(* PLC project IndraLogic.project, IndraLogic indralogic *)
(* stored: creationDateTime 2023-05-04T16:21:11.22622, modificationDateTime 2023-04-06T09:56:36 *)

{attribute 'symbol' := 'none'}
TYPE ST_ComBasketRotation : STRUCT
  fBasketRotationSpeed : REAL;  (* Drehzahl 0 <= x <= 4 l/min *)
  diagCodeBasketRotation : IL_INLN_DIAG_CODE;  (* Sensor-Diagnose: Temperatur *)
END_STRUCT;
END_TYPE

{attribute 'symbol' := 'readwrite'}
TYPE ST_TankErrorState : STRUCT
  bErrorTankLevelLow : BOOL;
  bErrorTankLevelFull : BOOL;
  bErrorFreshWaterSupply : BOOL;
  bErrorTankTemperatureCriticalLow : BOOL;
  bErrorTankTemperatureCriticalHigh : BOOL;
END_STRUCT;
END_TYPE

{attribute 'symbol' := 'none'}
TYPE ST_PowerMeasurementUMG96RM : STRUCT
  modeReturn : INT;  (* Die genaue Konfiguration ist dem Handbuch zu Janitza UMG96RM-P (ab S.82) zu entnehmen *)
  value : ARRAY[0..26] OF REAL;
  count : INT := 27;
  StromGes : REAL;
  WirkleistungGes : REAL;
  BlindleistungGes : REAL;
  Frequenz : REAL;
END_STRUCT;
END_TYPE

{attribute 'symbol' := 'readwrite'}
TYPE ST_SetKEAProgramManual : STRUCT
  fTankTemperatureSetPointManual : REAL;  (* Bereich: 30...75°C *)
  fTankHeaterHysteresisWidthManual : REAL;  (* Definiert Range der Tankheizung *)
  fAirHeatingTemperatureSetPointManual : REAL;  (* Bereich: 50...110°C *)
  fTemperatureLimitLowerWorking : REAL;  (* minimal temperature to start process *)
  fTemperatureLimitUpperWorking : REAL;  (* maximal temperature to start process *)
  nDurationSprayCleaningManual : INT;  (* Bereich: 0...300 Sekunden - Zeit für Schrittkette *)
  nDurationDrippingManual : INT;  (* Bereich: 0...300 Sekunden - Zeit für Schrittkette *)
  nDurationSuctionManual : INT;  (* Bereich: 0...300 Sekunden - Zeit für Schrittkette *)
  nDurationBlowingManual : INT;  (* Bereich: 0...300 Sekunden - Zeit für Schrittkette *)
  nDurationConvectionDryingManual : INT;  (* Bereich: 0...300 Sekunden - Zeit für Schrittkette *)
  bProgramWithBasketRotationManual : BOOL;
  bProgramWithBasketRotation : BOOL;  (* Keine Korbrotation *)
  sTypeWorkpiece : STRING;
  fMassWorkpiece : REAL;  (* mass in kg *)
END_STRUCT;
END_TYPE

{attribute 'symbol' := 'readwrite'}
TYPE ST_KEALocalSetParameters : STRUCT
  nSelectProgram : INT;
  bSetSelectedProgram : BOOL;
  bResetErrors : BOOL;
  bOpenDoor : BOOL;
  nWorkpieces : INT;
END_STRUCT;
END_TYPE

{attribute 'symbol' := 'readwrite'}
TYPE ST_StoreEnergyInherentlyState : STRUCT
  fNominalLoad : REAL;  (* static; module's nominal load *)
  sMachineStateCorrelation : STRING;  (* static; machine states in which the module can be used as inherent energy storage: oﬀ , standby , operational or working *)
  sProcessStepCorrelation : STRING;  (* static; process steps in which the module is active *)
  sPowerUnit : STRING;  (* static; unit of nominal load and power consumption *)
  bOperatingPoint : BOOL;  (* dynamic; module's switching state *)
  fProcessValue : REAL;  (* dynamic; process value influenced by the module *)
  aFlexibilityLimits : ARRAY[1..2] OF REAL;  (* dynamic; upper and lower limits in which the energy-ﬂexible module may operate *)
  sProcessValueUnit : STRING;  (* static; unit of process value and flexibility limits *)
END_STRUCT;
END_TYPE

{attribute 'symbol' := 'readwrite'}
TYPE ST_CleaningChamberState : STRUCT
  bPumpSupplyStatusOn : BOOL;
  bRotationBasketStatusOn : BOOL;
  bRotationBasketDirectionOfRotation : BOOL;
  bRotationNoozleFrameStatusOn : BOOL;
  bExhaustAirFanStatusOn : BOOL;
  bBlastNoozleTopStatusOn : BOOL;
  bBlastNoozleBottomStatusOn : BOOL;
  bProtectiveDoorLoadingOpen : BOOL;
END_STRUCT;
END_TYPE

{attribute 'symbol' := 'readwrite'}
TYPE ST_InterruptProcessState : STRUCT
  stepEnergyConsumption : ST_StepEnergyConsumption;  (* static; shows total energy consumption per step for all steps that can be interrupted *)
  sEnergyUnit : STRING;  (* static; unit of energy consumption *)
  fMachinePowerConsumption : REAL;  (* dynamic; current power consumption of the whole machine *)
  stepPowerConsumption : ST_StepPowerConsumption;  (* static; shows total power consumption per step for all energy relevant steps *)
  sPowerUnit : STRING;  (* static; unit of nmachine power consumption *)
  stepDuration : ST_StepDuration;
  sMachineState : STRING;  (* dynamic; shows current machine state: oﬀ , standby , operational or working *)
  fInterruptionCountdown : REAL;  (* dynamic; shows duration until the next position for process interruption is reached *)
  fInterruptionCountdownUnit : STRING;  (* static; unit of interruption countdown *)
  nInterruptedState : E_KEAOperatingState;  (* last state before interruption *)
END_STRUCT;
END_TYPE

{attribute 'qualified_only'}
{attribute 'strict'}
TYPE E_SystemControlState : (automatic := 0, algorithm := 1, manual := 2);
END_TYPE

{attribute 'qualified_only'}
{attribute 'strict'}
TYPE E_SystemOperatingState : (standby := 0, rampUp := 1, rampDown := 2, operational := 3, working := 4);
END_TYPE

{attribute 'symbol' := 'readwrite'}
TYPE ST_Control : STRUCT
  bSetStatusOnAlgorithm : BOOL;  (* turn actor on *)
  bSetStatusOnManual : BOOL;  (* turn actor on *)
  bAlgorithmModeActivated : BOOL;  (* activate algorithm control *)
  bManualModeActivated : BOOL;  (* activate manual control *)
END_STRUCT;
END_TYPE

{attribute 'symbol' := 'readwrite'}
TYPE ST_ControlState : STRUCT
  bStatusOn : BOOL;  (* status on / off *)
  sAccessMode : STRING;  (* current access mode as string *)
  nAccessmode : E_SystemControlState;  (* current access mode (1 = automatic, 2 = algorihm, 3 = manual) *)
END_STRUCT;
END_TYPE

{attribute 'symbol' := 'readwrite'}
TYPE ST_SensorState : STRUCT
  fValue : REAL;  (* status on / off *)
  sUnit : STRING;  (* current unit of sensor value *)
END_STRUCT;
END_TYPE

{attribute 'symbol' := 'readwrite'}
TYPE ST_SetPointState : STRUCT
  fOperatingPoint : REAL;  (* current operating point *)
  fSetPoint : REAL;  (* current set point *)
  sSetPointUnit : STRING;  (* current set point unit *)
  sOperatingPointUnit : STRING;  (* current operating point unit *)
  aSetPointLimits : ARRAY[1..2] OF REAL;  (* lower and upper limit of setpoint *)
END_STRUCT;
END_TYPE

{attribute 'symbol' := 'readwrite'}
TYPE ST_SetSetPoint : STRUCT
  fSetPointAlgorithm : REAL;  (* set setpoint in percent 0.0 - 100.0 *)
  fSetPointManual : REAL;  (* set setpoint in percent 0.0 - 100.0 *)
END_STRUCT;
END_TYPE

{attribute 'symbol' := 'readwrite'}
TYPE ST_SystemState : STRUCT
  sOperatingState : STRING;  (* operating state (standby, operational, working) *)
  nOperatingState : E_SystemOperatingState;  (* operating state (standby, operational, working) *)
  bError : BOOL;  (* true if there is an error in any system component *)
END_STRUCT;
END_TYPE

{attribute 'symbol' := 'readwrite'}
TYPE ST_InletAirHeatingErrorState : STRUCT
  bInletAirShutOffValveOpeningError : BOOL;
  bInletAirShutOffValveClosingError : BOOL;
  bInletAirShutOffValveSensorsError : BOOL;
  bInletAirFanError : BOOL;
  bAirSupplyTempSensorError : BOOL;
  bErrorAirTemperatureCriticalLow : BOOL;
  bErrorAirTemperatureCriticalHigh : BOOL;
END_STRUCT;
END_TYPE

{attribute 'symbol' := 'readwrite'}
TYPE ST_TempSensorState : STRUCT
  {attribute 'symbol' := 'none'}
  senTdiag : IL_INLN_DIAG_CODE;  (* Sensor-Diagnose: Temperatur *)
END_STRUCT;
END_TYPE

{attribute 'symbol' := 'readwrite'}
TYPE ST_TankState : STRUCT
  bTankHeatingOn : BOOL;
  bSupplyFreshWaterOn : BOOL;
  bOilSeparationOn : BOOL;
  fTankTemperature : REAL;
  bFilterMonitor : BOOL;
  bTankLevelMin : BOOL;
  bTankLevelNominal : BOOL;
  bTankLevelMax : BOOL;
  bOilSeparationLevelMax : BOOL;
  bDemineralOk : BOOL;
  fTankHeaterHysteresisWidth : REAL;
  fTemperatureLimitLowerWorking : REAL;
  fTemperatureLimitUpperWorking : REAL;
  fTemperatureLimitLowerCritical : REAL;
  fTemperatureLimitUpperCritical : REAL;
  sTemperatureUnit : STRING;
  fCleaningFluidSpecificHeatCapacity : REAL;
  sCleaningFluidSpecificHeatCapacityUnit : STRING;
  fCleaningFluidDensity : REAL;
  sCleaningFluidDensityUnit : STRING;
  fTankVolume : REAL;
  sTankVolumeUnit : STRING;
END_STRUCT;
END_TYPE

{attribute 'symbol' := 'readwrite'}
TYPE ST_InletAirHeatingState : STRUCT
  fAirSupplyTemperature : REAL;
  bInletAirShutOffValveOpen : BOOL;
  bInletAirShutOffValveClosed : BOOL;
  bAirSupplyTempOk : BOOL;
  bAirSupplyFlowOk : BOOL;
  fTemperatureLimitLowerCritical : REAL;
  fTemperatureLimitUpperCritical : REAL;
  bInletAirFanStatusOn : BOOL;
END_STRUCT;
END_TYPE

{attribute 'symbol' := 'none'}
TYPE ST_KEADefaultParameters : STRUCT
  tBlastNoozlesPulseDuration : TIME := TIME#200ms;  (* Bereich: 0,2...1,0 Sekunden *)
  tBlastNoozlesPulsePeriod : TIME := TIME#700ms;  (* Bereich: 0,2...1,0 Sekunden *)
  tBasketHomeingDuration : TIME := TIME#500ms;  (* Bereich: 0,000...2,000 Sekunden - in Millisekunden verarbeiten *)
  fBasketRotationSpeed : REAL := 3;  (* Bereich: 1.5...4.0 l/min - Vorgabe für Frequenzumrichter *)
  tMaxDurationExhaustFanOn : TIME := TIME#1m0s0ms;  (* Zeitliche Begrenzung Abluftgebläse wenn Tür offen *)
END_STRUCT;
END_TYPE

{attribute 'qualified_only'}
TYPE E_KEAOperatingState : (standby := 0, rampUp := 1, operational := 2, sprayCleaning := 3, dripping := 4, suction := 5, blowing := 6, convectionDrying := 7, homing := 8, interruption := 9, break := 10, error := 11);
END_TYPE

{attribute 'symbol' := 'readwrite'}
TYPE ST_KEAProgramState : STRUCT
  sActiveProgram : STRING;
  fTankTemperatureSetPoint : REAL;  (* Bereich: 30...75°C *)
  fTankHeaterHysteresisWidth : REAL;  (* Definiert Range der Tankheizung *)
  fTemperatureLimitLowerWorking : REAL;  (* minimal temperature to start process *)
  fTemperatureLimitUpperWorking : REAL;  (* maximal temperature to start process *)
  fAirHeatingTemperatureSetPoint : REAL;  (* Bereich: 50...110°C *)
  nDurationSprayCleaning : INT;  (* Bereich: 0...300 Sekunden - Zeit für Schrittkette *)
  nDurationDripping : INT;  (* Bereich: 0...300 Sekunden - Zeit für Schrittkette *)
  nDurationSuction : INT;  (* Bereich: 0...300 Sekunden - Zeit für Schrittkette *)
  nDurationBlowing : INT;  (* Bereich: 0...300 Sekunden - Zeit für Schrittkette *)
  nDurationConvectionDrying : INT;  (* Bereich: 0...300 Sekunden - Zeit für Schrittkette *)
  sDurationUnit : STRING;  (* duration unit = seconds *)
  bProgramWithBasketRotation : BOOL;
  sTypeWorkpiece : STRING;
  fMassWorkpiece : REAL;
  sMassWorkpieceUnit : STRING;
END_STRUCT;
END_TYPE

{attribute 'symbol' := 'readwrite'}
TYPE ST_KEAState : STRUCT
  sKEAOperatingState : STRING;  (* operating state (standby, operational, rampUp, working, sprayCleaning, dripping, suction, blowing, convectionDrying, homing, interruption) *)
  nKEAOperatingState : E_KEAOperatingState;  (* operating state (standby, operational, rampUp, working, sprayCleaning, dripping, suction, blowing, convectionDrying, homing, interruption) *)
  nWorkpieces : INT;
  fMassWorkpiece : REAL;
  fCurrent : REAL;
  fRealPower : REAL;
  fReactivePower : REAL;
  fFrequency : REAL;
END_STRUCT;
END_TYPE

{attribute 'symbol' := 'readwrite'}
TYPE ST_KEAErrorState : STRUCT
  bGlobalError : BOOL;
  bTankHeatingSystemError : BOOL;
  bInletAirHeatingSystemError : BOOL;
  bEmergencyStopError : BOOL;
  bConditionToStartError : BOOL;
END_STRUCT;
END_TYPE

{attribute 'symbol' := 'readwrite'}
TYPE ST_CleaningChamberErrorState : STRUCT
  bMotorsDrivesError : BOOL;
  bDoorLoadingSafetyError : BOOL;
END_STRUCT;
END_TYPE

{attribute 'symbol' := 'readwrite'}
TYPE ST_StepEnergyConsumption : STRUCT
  fEnergyConsumptionSprayCleaning : REAL;
  fEnergyConsumptionConvectionDrying : REAL;
END_STRUCT;
END_TYPE

{attribute 'symbol' := 'readwrite'}
TYPE ST_StepDuration : STRUCT
  fDurationSprayCleaning : REAL;
  fDurationDripping : REAL;
  fDurationSuction : REAL;
  fDurationBlowing : REAL;
  fDurationConvectionDrying : REAL;
  sDurationUnit : STRING;
END_STRUCT;
END_TYPE

{attribute 'symbol' := 'readwrite'}
TYPE ST_InterruptProcess : STRUCT
  bInterruptProcessAlgorithm : BOOL;  (* interrupt process *)
  bInterruptProcessManual : BOOL;  (* interrupt process *)
END_STRUCT;
END_TYPE

{attribute 'symbol' := 'readwrite'}
TYPE ST_StepPowerConsumption : STRUCT
  fPowerConsumptionSprayCleaning : REAL;
  fPowerConsumptionConvectionDrying : REAL;
  fPowerConsumptionBlowing : REAL;
  fPowerConsumptionDripping : REAL;
  fPowerConsumptionSuction : REAL;
  fPowerConsumptionHoming : REAL;
  fPowerConsumptionOperational : REAL;
END_STRUCT;
END_TYPE

VAR_GLOBAL  (* outputs *)
  bCPU_OK AT %QX10.0 : BOOL;  (* Freigabe: Immer - Immer EINS, da Rexroth Steuerung keine Verbindung zum HMI hat *)
  bTankHeatingOn AT %QX10.1 : BOOL;  (* Freigabe: Keine Stoerung - EIN wenn Tanktemperatur <= (Solltemp_Tank -2) - NULL wenn Tanktemperatur >= Solltemp_Tank *)
  bPumpSupplyOn AT %QX10.2 : BOOL;  (* Spritzpumpe, Freigabe: Keine Stoerung und Besch_Tuer_Gesch - EIN wenn von Schrittkette benötigt wird - NULL wenn Schritt== 0 *)
  bSupplyFreshWaterOn AT %QX10.3 : BOOL;  (* Freigabe: Keine Stoerung - EIN wenn (Schritt==0) UND (Sollniveau==Nachtanken=EINS) *)
  bOilSeparationOn AT %QX10.4 : BOOL;  (* Freigabe: Keine Stoerung und Oelabsch_Niveau==NULL und Niveau_Soll==0 - EIN während Reinigungsprogramm, ggf. mit Nachlauf - Beachte: Bei kalten Wasser und Chemiezusatz Schaumentwicklung, ggf. nur über 35°C betreiben (Temp.schaltpunkt mit Hysterese belegen) *)
  bRotationBasketEnable AT %QX10.5 : BOOL;  (* Freigabe: Keine Stoerung und Besch_Tuer_Gesch - EIN wenn von Schrittkette benötigt wird - NULL wenn Schritt== 0 *)
  bRotationBasketDirectionOfRotation AT %QX10.6 : BOOL;  (* Freigabe: Immer - EIN wenn von Schrittkette benötigt wird - NULL wenn von Schrittkette benötigt wird *)
  bRotationNoozleFrameEnable AT %QX10.7 : BOOL;  (* Freigabe: Keine Stoerung und Besch_Tuer_Gesch - EIN wenn von Schrittkette benötigt wird - NULL wenn Schritt== 0 *)
  bOpenProtectiveDoorLoading AT %QX11.0 : BOOL;  (* Freigabe: Kein Not-Halt - EIN wenn (Schritt==0) UND (Tuertaster==EINS) *)
  bExhaustAirFanOn AT %QX11.1 : BOOL;  (* Freigabe: Keine Stoerung und bDoorClosed - EIN wenn von Schrittkette benötigt wird - NULL wenn Schritt== 0 UND Besch_Tuer_Gesch *)
  bInletAirFanOn AT %QX11.2 : BOOL;  (* Freigabe: Keine Stoerung und bDoorClosed - EIN wenn von Schrittkette benötigt wird - NULL wenn Schritt== 0 *)
  bOpenInletAirShutOffValve AT %QX11.3 : BOOL;  (* Freigabe: Keine Stoerung und bDoorClosed - EIN wenn von Schrittkette benötigt wird - NULL wenn Schritt== 0 *)
  bInletAirHeaterOn AT %QX11.4 : BOOL;  (* Freigabe: Keine Stoerung und bDoorClosed - EIN wenn von Schrittkette benötigt wird - NULL wenn Schritt== 0 *)
  bBlastNoozleTopOn AT %QX11.5 : BOOL;  (* Freigabe: Keine Stoerung und bDoorClosed - EIN wenn von Schrittkette benötigt wird; s. Pulssteuerung - NULL wenn Schritt== 0 *)
  bBlastNoozleBottomOn AT %QX11.6 : BOOL;  (* Freigabe: Keine Stoerung und bDoorClosed - EIN wenn von Schrittkette benötigt wird; s. Pulssteuerung - NULL wenn Schritt== 0 *)
END_VAR

VAR_GLOBAL  (* inputs - -----Variablen die die Maschine an die Steuerung meldet--- *)
  bStartButton AT %IX0.1 : BOOL;  (* EINS wenn gedrückt *)
  bFilterMonitor AT %IX10.0 : BOOL;  (* Meldung, Warnung wenn NULL und Spritzpumpe EIN - Verzoegerung 10 sec *)
  bTankLevelMin_NOT AT %IX10.1 : BOOL;  (* Meldung, Stoerung wenn NULL - Verzoegerung 3 sec *)
  bTankLevelNominal_NOT AT %IX10.2 : BOOL;  (* NULL: Niveau OK; EINS: Nachtanken *)
  bTankLevelMax_NOT AT %IX10.3 : BOOL;  (* Meldung, Stoerung wenn NULL - Verzoegerung 3 sec *)
  bOilSeparationLevelMax AT %IX10.4 : BOOL;  (* Meldung, Warnung wenn EINS - Verzoegerung 10 sec *)
  bBasketHomed AT %IX10.5 : BOOL;  (* EINS wenn Antrieb Korb in Nulllage *)
  bDoorClosed AT %IX10.6 : BOOL;  (* EINS wenn Tuer geschlossen *)
  bNoozleFrameHomed AT %IX10.7 : BOOL;  (* EINS wenn Antrieb Duesen in Nulllage *)
  bInletAirShutOffValveOpen AT %IX11.1 : BOOL;  (* Meldung, Stoerung wenn NULL und Zuluftklappe EIN - Verzoegerung 5 sec *)
  bInletAirShutOffValveClosed AT %IX11.2 : BOOL;  (* Meldung, Stoerung wenn NULL und Zuluftklappe AUS - Verzoegerung 5 sec *)
  bAirSupplyTempSensorOk AT %IX11.3 : BOOL;  (* Meldung, Stoerung wenn NULL - Verzoegerung 1 sec *)
  bAirSupplyFlowOk AT %IX11.4 : BOOL;  (* Meldung, Stoerung wenn NULL und Zuluftgeblaese EIN - Verzogerung 20 sec *)
  bDemineralOk AT %IX11.7 : BOOL;  (* Meldung, Stoerung wenn NULL und Frischwasser EIN - Verzogerung 5 sec *)
  bEmergencyStopOk AT %IX0.0 : BOOL;  (* Meldung, Stoerung wenn NULL - Verzoegerung 0 sec *)
  bMotorsDrivesOk AT %IX0.3 : BOOL;  (* Meldung, Stoerung wenn NULL - Verzoegerung 0 sec *)
  bConditionToStartOk AT %IX0.4 : BOOL;  (* Meldung, Stoerung wenn NULL - Verzoegerung 0 sec (Quittierung Nothalt drücken, damit ok) *)
  bDoorLoadingSafetyOk AT %IX0.6 : BOOL;  (* Meldung, Stoerung wenn NULL - Verzoegerung 0 sec *)
END_VAR

INTERFACE ITF_ActorContinous
METHOD SetSetPointLimits : BOOL
END_METHOD
END_INTERFACE

INTERFACE ITF_System
METHOD RampDown : BOOL
  VAR_OUTPUT
    bRampDownFinished : BOOL := FALSE;
  END_VAR
END_METHOD
METHOD Operational : BOOL
  VAR_OUTPUT
    bSwitchToWorking : BOOL := FALSE;
  END_VAR
END_METHOD
METHOD CheckError : BOOL
  VAR_OUTPUT
    bError : BOOL;
  END_VAR
END_METHOD
METHOD Working : BOOL
  VAR_OUTPUT
    bSwitchToOperational : BOOL := FALSE;
  END_VAR
END_METHOD
METHOD RampUp : BOOL
  VAR_OUTPUT
    bRampUpFinished : BOOL := FALSE;
  END_VAR
END_METHOD
METHOD Standby : BOOL
END_METHOD
METHOD SystemFlowControl : INT
END_METHOD
END_INTERFACE

{attribute 'symbol' := 'none'}
PROGRAM PRG_AnalogInputs
  VAR
    fbAI3 : IL_AI8SfIs;
    wInProcessData : ARRAY[0..1] OF WORD;
    wOutProcessData : ARRAY[0..1] OF WORD;
  END_VAR
  VAR_OUTPUT
    tankTempSensor : ST_TempSensorState;
    airSupplyTempSensor : ST_TempSensorState;
  END_VAR

            // Konfiguration (Tempertur Sensoren 4...20 mA)

//Tanktemperatur
fbAI3.ChannelConfig[0].InputRange 	:= IL_INLN_AI_RANGE.UNIPOLAR4TO20MA;
fbAI3.ChannelConfig[0].HighLimit 	:= REAL#100.0;		// 100°C
fbAI3.ChannelConfig[0].LowLimit   	:= REAL#0.0;		// 0°C
fbAI3.ChannelConfig[0].NoOfSamples 	:= BYTE#16;

//Zulufttemperatur
fbAI3.ChannelConfig[1].InputRange 	:= IL_INLN_AI_RANGE.UNIPOLAR4TO20MA;
fbAI3.ChannelConfig[1].HighLimit 	:= REAL#300.0;		// 300°C
fbAI3.ChannelConfig[1].LowLimit   	:= REAL#0.0;		// 0°C
fbAI3.ChannelConfig[1].NoOfSamples 	:= BYTE#16;




fbAI3.ChannelSelect                	:= BYTE#2#00000111;
fbAI3.InProcData_0                 	:= wInProcessData[0];
fbAI3.InProcData_1                 	:= wInProcessData[1];
wOutProcessData[0]                  := fbAI3.OutProcData_0;
wOutProcessData[1]                  := fbAI3.OutProcData_1; 

// FB-Aufruf
fbAI3(Enable :=TRUE);

// Daten lesen
IF fbAI3.InOperation = TRUE THEN	
	//neu:
	// Normalisierte Werte speichern
	tankTempSensor.fValue		:= fbAI3.OutputData[0].NormalizedValue;
	airSupplyTempSensor.fValue	:= fbAI3.OutputData[1].NormalizedValue;
	
	// set sensor value unit
	tankTempSensor.sUnit 		:= 'degreeC';
	airSupplyTempSensor.sUnit 	:= 'degreeC';
	
	// Diagnose-Codes speichern
	tankTempSensor.senTdiag			:= fbAI3.OutputData[0].DiagCode;
	airSupplyTempSensor.senTdiag	:= fbAI3.OutputData[1].DiagCode;
END_IF

          
END_PROGRAM

PROGRAM Plc_Main
  VAR
    KEA : FB_KEASystem;
  END_VAR

            (* vvvvvvvvvvvvvvvvvvvvvvvvvvvv nicht ändern vvvvvvvvvvvvvvvvvvvvvvvvvvvv *)

(*------------------ Errors & Warnings -------------*)
//PRG_Errors();
//PRG_Warnings();

(*------------------ Input / Output Mapping -------------*)
PRG_AnalogInputs();
PRG_AnalogOutputs();
prLeistungsmessungUMG();
(*------------------ Cleaning program -------------*)
KEA(bSetStatusOnAutomatic := TRUE);
          
END_PROGRAM

{attribute 'symbol' := 'none'}
PROGRAM PRG_AnalogOutputs
  VAR_INPUT
    comBasketRotation : ST_ComBasketRotation;
  END_VAR
  VAR
    fbAO1 : IL_AO2SfBp;
    wInProcessData : ARRAY[0..1] OF WORD;
    wOutProcessData : ARRAY[0..1] OF WORD;
  END_VAR

            // Konfiguration (Drehzahl_Antr_Korb)
fbAO1.ModuleType := IL_INLN_SF_BP.BPUNIPOLAR10V;
fbAO1.ResetOutput := TRUE;
fbAO1.NonVolatile := TRUE;
fbAO1.InputData[0].HighLimit := REAL#4.0;
fbAO1.InputData[0].LowLimit := REAL#0.0;
fbAO1.ChannelSelect := BYTE#2#00000001;
fbAO1.InProcData_0 := wInProcessData[0];
fbAO1.InProcData_1 := wInProcessData[1];
wOutProcessData[0] := fbAO1.OutProcData_0 ;
wOutProcessData[1] := fbAO1.OutProcData_1 ;

// FB-Aufruf
fbAO1(Enable :=TRUE);

// Daten ausgeben
(* Sobald der FB arbeitet, beginnt er sein Spannungs- bzw. Stromsignal zu erzeugen.   
Die Ausgabe variiert dabei entsprechend dem Wert am 'Normalized value'-Eingang.*)
IF fbAO1.InOperation = TRUE THEN
	// Normalisierte Werte ausgeben
	fbAO1.InputData[0].NormalizedValue := comBasketRotation.fBasketRotationSpeed;
		
	// Diagnose-Codes speichern
	comBasketRotation.diagCodeBasketRotation := fbAO1.DiagCode_0;
END_IF

          
END_PROGRAM

{attribute 'symbol' := 'none'}
PROGRAM prLeistungsmessungUMG
  VAR_OUTPUT
    LeistungsmessungUMG : ST_PowerMeasurementUMG96RM;
  END_VAR
  VAR
    mode AT %QB14 : BYTE;
    wInProcessData AT %IW14 : ARRAY[0..124] OF BYTE;
  END_VAR
  VAR
    modeLeistungsmessungUMG : BYTE := 8;
    i : INT;
    prozesswort : DWORD;
    pointR : POINTER TO REAL;
  END_VAR

            mode := modeLeistungsmessungUMG;
LeistungsmessungUMG.modeReturn := BYTE_TO_INT(wInProcessData[1]);

IF (i < (LeistungsmessungUMG.count))THEN
	prozesswort := SHL(BYTE_TO_DWORD(wInProcessData[(0+(4*i))]), 24) OR SHL(BYTE_TO_DWORD(wInProcessData[(3+(4*i))]), 16) OR SHL(BYTE_TO_DWORD(wInProcessData[(2+(4*i))]), 8) OR BYTE_TO_DWORD(wInProcessData[(5+(4*i))]);
	pointR := ADR(prozesswort);
	LeistungsmessungUMG.value[i] := pointR^;
	LeistungsmessungUMG.StromGes := LeistungsmessungUMG.value[10];
	LeistungsmessungUMG.WirkleistungGes  := LeistungsmessungUMG.value[18];
	LeistungsmessungUMG.BlindleistungGes  := LeistungsmessungUMG.value[19];
	LeistungsmessungUMG.Frequenz  := LeistungsmessungUMG.value[17];
	i := i+1;
ELSE
	i :=0;
END_IF
          
END_PROGRAM

{attribute 'symbol' := 'none'}
FUNCTION_BLOCK FB_Actor2Point
  VAR_INPUT
    bSetStatusOnAutomatic : BOOL;  (* turn actor on *)
    bAlgorithmPermission : BOOL;  (* is true if control by algorithm is allowed *)
  END_VAR
  VAR
    {attribute 'symbol' := 'readwrite'}
    control : ST_Control;
    {attribute 'symbol' := 'readwrite'}
    controlState : ST_ControlState;
    bSetStatusOn : BOOL;  (* actual internal value to switch on *)
  END_VAR

            SelectControlMode();
controlState.bStatusOn := bSetStatusOn;
          

METHOD SelectControlMode : BOOL
                  //change access mode
IF control.bManualModeActivated THEN
	controlState.nAccessmode := E_SystemControlState.manual;
	controlState.sAccessMode := 'manual';
	bSetStatusOn := control.bSetStatusOnManual;
ELSIF control.bAlgorithmModeActivated AND bAlgorithmPermission THEN
	controlState.nAccessmode := E_SystemControlState.algorithm;
	controlState.sAccessMode := 'algorithm';
	bSetStatusOn := control.bSetStatusOnAlgorithm;
ELSE
	controlState.nAccessmode := E_SystemControlState.automatic;
	controlState.sAccessMode := 'automatic';
	bSetStatusOn := bSetStatusOnAutomatic;
END_IF
                
END_METHOD

PROPERTY bStatusOn : BOOL
GET
                    bStatusOn := bSetStatusOn;
                  
END_GET
END_PROPERTY
END_FUNCTION_BLOCK

{attribute 'symbol' := 'none'}
FUNCTION_BLOCK FB_Sensor
  VAR
    {attribute 'symbol' := 'readwrite'}
    sensorState : ST_SensorState;
  END_VAR

            
          
END_FUNCTION_BLOCK

{attribute 'symbol' := 'none'}
FUNCTION_BLOCK FB_KEASystem EXTENDS FB_System2Point IMPLEMENTS ITF_System
  VAR
    {attribute 'symbol' := 'readwrite'}
    tank : FB_TankSystem;  (* subsystems *)
    {attribute 'symbol' := 'readwrite'}
    inletAirHeating : FB_InletAirHeatingSystem;
    {attribute 'symbol' := 'readwrite'}
    cleaningChamber : FB_CleaningChamberSystem;
    bStartButton : BOOL;  (* sensors *)
    bEmergencyStopOk : BOOL;
    bConditionToStartOk : BOOL;
    UMG96RM_powerMeasurement : ST_PowerMeasurementUMG96RM;
    localDefaultParameters : ST_KEADefaultParameters;  (* default parameters *)
    {attribute 'symbol' := 'readwrite'}
    localState : ST_KEAState;  (* states *)
    {attribute 'symbol' := 'readwrite'}
    errorState : ST_KEAErrorState;
    {attribute 'symbol' := 'readwrite'}
    programState : ST_KEAProgramState;
    {attribute 'symbol' := 'readwrite'}
    localSetParameters : ST_KEALocalSetParameters;  (* parameter sets *)
    {attribute 'symbol' := 'readwrite'}
    setKEAProgramManual : ST_SetKEAProgramManual;
    bInterruptProcess : BOOL := FALSE;  (* interruption *)
    {attribute 'symbol' := 'readwrite'}
    interruptProcess : ST_InterruptProcess;
    {attribute 'symbol' := 'readwrite'}
    interruptProcessState : ST_InterruptProcessState;
    bGlobalError : BOOL;  (* local variables *)
    tBlastNoozlesPulseDuration : TIME := localDefaultParameters.tBlastNoozlesPulseDuration;
    tBlastNoozlesPulsePeriod : TIME := localDefaultParameters.tBlastNoozlesPulsePeriod;
    tBasketHomeingDuration : TIME := localDefaultParameters.tBasketHomeingDuration;
    fBasketRotationSpeed : REAL := localDefaultParameters.fBasketRotationSpeed;
    tMaxDurationExhaustFanOn : TIME := localDefaultParameters.tMaxDurationExhaustFanOn;
    tTimeToNextInterruption : TIME;
    nWorkpieces : INT;  (* number of workpieces in tray *)
    fCurrent : REAL;
    fRealPower : REAL;
    fReactivePower : REAL;
    fFrequency : REAL;
    bStartExhaustFan : BOOL;
    nSelectProgram : INT := 1;  (* standard program 1 : Arepron *)
    bSetSelectedProgram : BOOL;
    bResetErrors : BOOL;
    bOpenDoor : BOOL;
    sActiveProgram : STRING;  (* state *)
    fTankTemperatureSetPoint : REAL;  (* Bereich: 30...75°C *)
    fTankHeaterHysteresisWidth : REAL;  (* Definiert Range der Tankheizung *)
    fAirHeatingTemperatureSetPoint : REAL;  (* Bereich: 50...110°C *)
    fTemperatureLimitLowerWorking : REAL;  (* minimal tempereture to start process *)
    fTemperatureLimitUpperWorking : REAL;  (* maximal tempereture to start process *)
    tDurationSprayCleaning : TIME;  (* Bereich: 0...300 Sekunden - Zeit für Schrittkette *)
    tDurationDripping : TIME;  (* Bereich: 0...300 Sekunden - Zeit für Schrittkette *)
    tDurationSuction : TIME;  (* Bereich: 0...300 Sekunden - Zeit für Schrittkette *)
    tDurationBlowing : TIME;  (* Bereich: 0...300 Sekunden - Zeit für Schrittkette *)
    tDurationConvectionDrying : TIME;  (* Bereich: 0...300 Sekunden - Zeit für Schrittkette *)
    bProgramWithBasketRotation : BOOL;
    sTypeWorkpiece : STRING;
    fMassWorkpiece : REAL;
  END_VAR

            MAIN();
ReadInputs();
SelectProgram();
SelectInterruptionMode();

// Algorithm has permission if KEA is not in error state
bAlgorithmPermission := NOT bGlobalError;

// instantiate submodels
tank(
	bGlobalError					:= bGlobalError,
	bResetErrors					:= bResetErrors,
	bAlgorithmPermission 			:= TRUE, 
	fSetPointAutomatic 				:= fTankTemperatureSetPoint, 
	fTankHeaterHysteresisWidth 		:= fTankHeaterHysteresisWidth,
	fTemperatureLimitLowerWorking 	:= fTemperatureLimitLowerWorking,
	fTemperatureLimitUpperWorking 	:= fTemperatureLimitUpperWorking
);
inletAirHeating(
	bGlobalError			:= bGlobalError,
	bResetErrors			:= bResetErrors,
	bAlgorithmPermission 	:= TRUE, 
	fSetPointAutomatic 		:= fAirHeatingTemperatureSetPoint
);
cleaningChamber(
	bGlobalError 				:= bGlobalError,
	bResetErrors				:= bResetErrors,
	tMaxDurationExhaustFanOn 	:= tMaxDurationExhaustFanOn
);
// set states
SetStates();

// set ouputs
outputs.bCPU_OK := TRUE;
PRG_AnalogOutputs.comBasketRotation.fBasketRotationSpeed := fBasketRotationSpeed;
          

METHOD StartButtonEdgeDetection : BOOL
  VAR_INPUT
    bButton : BOOL;
  END_VAR
                  RisingEdge(CLK := bButton, Q => StartButtonEdgeDetection);
                
END_METHOD

METHOD ReadInputs : BOOL
                  // read sensors
bStartButton 		:= StartButtonEdgeDetection(inputs.bStartButton);
bEmergencyStopOk 	:= inputs.bEmergencyStopOk;
bConditionToStartOk	:= inputs.bConditionToStartOk;

// read from umg 96 rm
fCurrent 		:= prLeistungsmessungUMG.LeistungsmessungUMG.StromGes;
fRealPower 		:= prLeistungsmessungUMG.LeistungsmessungUMG.WirkleistungGes;
fReactivePower 	:= prLeistungsmessungUMG.LeistungsmessungUMG.BlindleistungGes;
fFrequency 		:= prLeistungsmessungUMG.LeistungsmessungUMG.Frequenz;

// read from opc ua
bResetErrors		:= localSetParameters.bResetErrors OR bStartButton;
bOpenDoor			:= localSetParameters.bOpenDoor;
bSetSelectedProgram := localSetParameters.bSetSelectedProgram;
IF bSetSelectedProgram THEN
	nSelectProgram	:= localSetParameters.nSelectProgram;
END_IF
nWorkpieces			:= localSetParameters.nWorkpieces;
                
END_METHOD

METHOD Standby : BOOL
                  // turn all cleaning chamber actors off
CleaningChamber.bPumpSupplyOn						:= FALSE;
CleaningChamber.bRotationBasketEnable 				:= FALSE;
CleaningChamber.bRotationBasketDirectionOfRotation 	:= FALSE;
CleaningChamber.bRotationNoozleFrameEnable 			:= FALSE;
CleaningChamber.bBlastNoozleTopOn					:= FALSE;
CleaningChamber.bBlastNoozleBottomOn				:= FALSE;

// turn off air heating
inletAirHeating.bSetStatusOnAutomatic := FALSE;

// turn off tank heating
tank.bSetStatusOnAutomatic := FALSE;

// open door if wanted
CleaningChamber.OpenDoor(
	bOpenDoor := bOpenDoor, 
	bInletAirHeaterOnStatus := inletAirHeating.bInletAirHeaterOn, 
	nActiveState := systemState.nOperatingState
);
                
END_METHOD

METHOD SprayCleaning : BOOL
                  // turn on pump, basket rotation if wanted and noozle frame
CleaningChamber.bPumpSupplyOn						:= TRUE;
CleaningChamber.bRotationBasketEnable 				:= bProgramWithBasketRotation;
CleaningChamber.bRotationBasketDirectionOfRotation 	:= FALSE;
CleaningChamber.bRotationNoozleFrameEnable 			:= TRUE;
CleaningChamber.bExhaustAirFanOn 					:= FALSE;
CleaningChamber.bBlastNoozleTopOn					:= FALSE;
CleaningChamber.bBlastNoozleBottomOn				:= FALSE;

// turn off air heating
inletAirHeating.bSetStatusOnAutomatic := FALSE;

// turn on tank heating
tank.bSetStatusOnAutomatic := TRUE;
                
END_METHOD

METHOD Dripping : BOOL
                  // turn on basket rotation if wanted, invert rotation
CleaningChamber.bPumpSupplyOn						:= FALSE;
CleaningChamber.bRotationBasketEnable 				:= bProgramWithBasketRotation;
CleaningChamber.bRotationBasketDirectionOfRotation 	:= TRUE;
CleaningChamber.bRotationNoozleFrameEnable 			:= FALSE;
CleaningChamber.bExhaustAirFanOn 					:= FALSE;
CleaningChamber.bBlastNoozleTopOn					:= FALSE;
CleaningChamber.bBlastNoozleBottomOn				:= FALSE;

// turn off air heating
inletAirHeating.bSetStatusOnAutomatic := FALSE;

// turn on tank heating
tank.bSetStatusOnAutomatic := TRUE;
                
END_METHOD

METHOD Suction : BOOL
                  // turn on basket rotation if wanted, invert rotation to normal, turn on exhaust air fan
CleaningChamber.bPumpSupplyOn						:= FALSE;
CleaningChamber.bRotationBasketEnable 				:= bProgramWithBasketRotation;
CleaningChamber.bRotationBasketDirectionOfRotation 	:= FALSE;
CleaningChamber.bRotationNoozleFrameEnable 			:= FALSE;
CleaningChamber.bExhaustAirFanOn 					:= TRUE;
CleaningChamber.bBlastNoozleTopOn					:= FALSE;
CleaningChamber.bBlastNoozleBottomOn				:= FALSE;

// turn off air heating
inletAirHeating.bSetStatusOnAutomatic := FALSE;

// turn on tank heating
tank.bSetStatusOnAutomatic := TRUE;
                
END_METHOD

METHOD Blowing : BOOL
  VAR
    bBlastNoozleBottomOn : BOOL;
    bBlastNoozleTopOn : BOOL;
  END_VAR
                  // call blast noozle control method
CleaningChamber.CtrlBlastNoozles(
	tBlastNoozlesPulseDuration := tBlastNoozlesPulseDuration,
	tBlastNoozlesPulsePeriod := tBlastNoozlesPulsePeriod,
	bBlastNoozleBottomOn => bBlastNoozleBottomOn, 
	bBlastNoozleTopOn => bBlastNoozleTopOn
);

// control blast noozles
CleaningChamber.bPumpSupplyOn						:= FALSE;
CleaningChamber.bRotationBasketEnable 				:= bProgramWithBasketRotation;
CleaningChamber.bRotationBasketDirectionOfRotation 	:= FALSE;
CleaningChamber.bRotationNoozleFrameEnable 			:= FALSE;
CleaningChamber.bExhaustAirFanOn 					:= TRUE;
CleaningChamber.bBlastNoozleBottomOn				:= bBlastNoozleBottomOn;
CleaningChamber.bBlastNoozleTopOn					:= bBlastNoozleTopOn;

// turn off air heating
inletAirHeating.bSetStatusOnAutomatic := FALSE;

// turn on tank heating
tank.bSetStatusOnAutomatic := TRUE;
                
END_METHOD

METHOD ConvectionDrying : BOOL
                  // turn on basket rotation if wanted, invert rotation to normal, turn on exhaust air fan
CleaningChamber.bPumpSupplyOn						:= FALSE;
CleaningChamber.bRotationBasketEnable 				:= bProgramWithBasketRotation;
CleaningChamber.bRotationBasketDirectionOfRotation 	:= FALSE;
CleaningChamber.bRotationNoozleFrameEnable 			:= FALSE;
CleaningChamber.bExhaustAirFanOn 					:= TRUE;
CleaningChamber.bBlastNoozleTopOn					:= FALSE;
CleaningChamber.bBlastNoozleBottomOn				:= FALSE;

// turn on air heating
inletAirHeating.bSetStatusOnAutomatic := TRUE;

// turn on tank heating
tank.bSetStatusOnAutomatic := TRUE;
                
END_METHOD

METHOD Homing : BOOL
  VAR_INPUT
    bNotOpenDoorAfterHoming : BOOL;
  END_VAR
  VAR_OUTPUT
    bHomingFinished : BOOL := FALSE;
  END_VAR
  VAR
    rTrigPositiveEdgeBasketHomed : R_TRIG;
    rTrigPositiveEdgeFrameHomed : R_TRIG;
  END_VAR
                  IF NOT bHomingStarted THEN
	fBasketRotationSpeedOld := fBasketRotationSpeed;
	bHomingStarted 			:= TRUE;
	nBasketHomingState 		:= 1;
	bBasketHomingFinished	:= FALSE;
END_IF 

// detect homing of basket and noozle frame
rTrigPositiveEdgeBasketHomed(CLK := CleaningChamber.bBasketHomed);
rTrigPositiveEdgeFrameHomed(CLK := CleaningChamber.bNoozleFrameHomed);

// basket homeing has to continue for a few seconds
tofDelayBasketHomeing(IN := rTrigPositiveEdgeBasketHomed.Q, PT := tBasketHomeingDuration);

CASE nBasketHomingState OF
	1: // normal homing
		bBasketHoming 			:= TRUE;
		// normal direction of basket rotation 
		cleaningChamber.bRotationBasketDirectionOfRotation := FALSE;
		IF rTrigPositiveEdgeBasketHomed.Q THEN
			nBasketHomingState := 2;
		END_IF
	2: // homing delay
		bBasketHoming := TRUE;
		// invert direction of basket rotation 
		cleaningChamber.bRotationBasketDirectionOfRotation := TRUE;
		IF NOT tofDelayBasketHomeing.Q THEN
			bBasketHomingFinished := TRUE;
			nBasketHomingState := 3;
		END_IF
	3: // homing finished
		bBasketHoming 			:= FALSE;
		// normal direction of basket rotation 
		cleaningChamber.bRotationBasketDirectionOfRotation := FALSE;
END_CASE

// turn off air heating
inletAirHeating.bSetStatusOnAutomatic := FALSE;

// turn on tank heating
tank.bSetStatusOnAutomatic := TRUE;

// if basket and noozle frame are finished stop rotation, reset basket rotation speed and direction and terminate homing
IF bBasketHomingFinished AND rTrigPositiveEdgeFrameHomed.Q THEN
	CleaningChamber.bRotationBasketEnable 				:= FALSE;
	CleaningChamber.bRotationNoozleFrameEnable			:= FALSE;
	fBasketRotationSpeed								:= fBasketRotationSpeedOld;
	cleaningChamber.bRotationBasketDirectionOfRotation 	:= FALSE;
	bHomingStarted										:= FALSE;
	bHomingFinished 									:= TRUE;
	// open door only if in normal homing state not after error
	IF NOT bNotOpenDoorAfterHoming THEN
		CleaningChamber.OpenDoor(
			bOpenDoor := TRUE, 
			bInletAirHeaterOnStatus := inletAirHeating.bInletAirHeaterOn, 
			nActiveState := E_SystemOperatingState.operational
		);
	END_IF
ELSE
	// else operate homing with slow basket rotation
	CleaningChamber.bRotationBasketEnable 		:= bBasketHoming;
	CleaningChamber.bRotationNoozleFrameEnable 	:= NOT rTrigPositiveEdgeFrameHomed.Q;
	fBasketRotationSpeed 						:= 1;
END_IF

// turn off other actors
CleaningChamber.bPumpSupplyOn						:= FALSE;
CleaningChamber.bBlastNoozleTopOn					:= FALSE;
CleaningChamber.bBlastNoozleBottomOn				:= FALSE;

                
END_METHOD

METHOD SystemFlowControl : INT
                  CheckError(bError => bSystemError);
systemState.bError := bSystemError;
TimeToNextInterruption(nKEAState := nKEAState, tStepElapsedTime := tStepElapsedTime);
tonStepTimer(Q => bSwitchState);

// reset remaining step time to zero when step is finished
IF bSwitchState THEN
	tStepTimeRemaining := T#0S;
END_IF

IF bSystemError THEN
	nKEAState := E_KEAOperatingState.error;
END_IF

CASE nKEAState OF
	E_KEAOperatingState.standby:
		nState := E_SystemOperatingState.standby;
		systemState.sOperatingState := 'standby';
		localState.sKEAOperatingState := 'standby';
		Standby();
		bSwitchState := FALSE;
		//if turned on switch to ramp-up
		IF(bSetStatusOn) THEN
			nKEAState := E_KEAOperatingState.rampUp;
		END_IF
	E_KEAOperatingState.rampUp:
		nState := E_SystemOperatingState.rampUp;
		systemState.sOperatingState := 'ramp-up';
		localState.sKEAOperatingState := 'ramp-up';
		RampUp(bRampUpFinished => bSwitchState);
		//if turned off switch to stand by
		IF(NOT bSetStatusOn) THEN
			nKEAState := E_KEAOperatingState.standby;
		//if ramp-up finished switch to operational
		ELSIF(bSwitchState) THEN
			nKEAState := E_KEAOperatingState.operational;
		END_IF
	E_KEAOperatingState.operational:
		nState := E_SystemOperatingState.operational;
		systemState.sOperatingState := 'operational';
		localState.sKEAOperatingState := 'operational';
		Operational(bSwitchToWorking => bSwitchState);
		//if turned off switch to stand-by
		IF(NOT bSetStatusOn) THEN
			nKEAState := E_KEAOperatingState.standby;
		ELSIF(bSwitchState) THEN
			// switch to interruption if interrupted
			IF(bInterruptProcess) THEN
				nInterruptedState := nKEAState;
				nKEAState := E_KEAOperatingState.interruption;
			// switch to sprayCleaning if desired
			ELSE
			nKEAState := E_KEAOperatingState.sprayCleaning;
			END_IF
		END_IF
	E_KEAOperatingState.sprayCleaning:
		nState := E_SystemOperatingState.working;
		systemState.sOperatingState := 'working';
		localState.sKEAOperatingState := 'working - spray cleaning';
		tonStepTimer(IN := TRUE, PT := tDurationSprayCleaning - tStepTimeRemaining, Q => bSwitchState, ET => tStepElapsedTime);
		SprayCleaning();
		// pause process step if button is pushed
		IF bStartButton THEN
			nStateInBreak := nKEAState;
			nKEAState := E_KEAOperatingState.break;
		//if cleaning is finished switch to dripping
		ELSIF(bSwitchState) THEN
			tonStepTimer.IN := FALSE;
			nKEAState := E_KEAOperatingState.dripping;
		END_IF
	E_KEAOperatingState.dripping:
		nState := E_SystemOperatingState.working;
		systemState.sOperatingState := 'working';
		localState.sKEAOperatingState := 'working - dripping';
		tonStepTimer(IN := TRUE, PT := tDurationDripping - tStepTimeRemaining, Q => bSwitchState, ET => tStepElapsedTime);
		Dripping();
		// pause process step if button is pushed
		IF bStartButton THEN
			nStateInBreak := nKEAState;
			nKEAState := E_KEAOperatingState.break;
		//if dripping is finished switch to suction
		ELSIF(bSwitchState) THEN
			tonStepTimer.IN := FALSE;
			nKEAState := E_KEAOperatingState.suction;
		END_IF
	E_KEAOperatingState.suction:
		nState := E_SystemOperatingState.working;
		systemState.sOperatingState := 'working';
		localState.sKEAOperatingState := 'working - suction';
		tonStepTimer(IN := TRUE, PT := tDurationSuction - tStepTimeRemaining, Q => bSwitchState, ET => tStepElapsedTime);
		Suction();
		// pause process step if button is pushed
		IF bStartButton THEN
			nStateInBreak := nKEAState;
			nKEAState := E_KEAOperatingState.break;
		//if suction is finished switch to blowing
		ELSIF(bSwitchState) THEN
			tonStepTimer.IN := FALSE;
			nKEAState := E_KEAOperatingState.blowing;
		END_IF
	E_KEAOperatingState.blowing:
		nState := E_SystemOperatingState.working;
		systemState.sOperatingState := 'working';
		localState.sKEAOperatingState := 'working - blowing';
		tonStepTimer(IN := TRUE, PT := tDurationBlowing - tStepTimeRemaining, Q => bSwitchState, ET => tStepElapsedTime);
		Blowing();
		// pause process step if button is pushed
		IF bStartButton THEN
			nStateInBreak := nKEAState;
			nKEAState := E_KEAOperatingState.break;
		ELSIF(bSwitchState) THEN
			// switch to interruption if interrupted
			IF(bInterruptProcess) THEN
				nInterruptedState := nKEAState;
				nKEAState := E_KEAOperatingState.interruption;
			//if blowing is finished switch to convection drying
			ELSE
			tonStepTimer.IN := FALSE;
			nKEAState := E_KEAOperatingState.convectionDrying;
			END_IF
		END_IF
	E_KEAOperatingState.convectionDrying:
		nState := E_SystemOperatingState.working;
		systemState.sOperatingState := 'working';
		localState.sKEAOperatingState := 'working - convection drying';
		tonStepTimer(IN := TRUE, PT := tDurationConvectionDrying - tStepTimeRemaining, Q => bSwitchState, ET => tStepElapsedTime);
		ConvectionDrying();
		// pause process step if button is pushed
		IF bStartButton THEN
			nStateInBreak := nKEAState;
			nKEAState := E_KEAOperatingState.break;
		//if convection drying is finished switch to homing
		ELSIF(bSwitchState) THEN
			tonStepTimer.IN := FALSE;
			nKEAState := E_KEAOperatingState.homing;
		END_IF
	E_KEAOperatingState.homing:
		nState := E_SystemOperatingState.working;
		systemState.sOperatingState := 'working';
		localState.sKEAOperatingState := 'working - homing';
		Homing(bNotOpenDoorAfterHoming := bErrorResetHoming, bHomingFinished => bSwitchState);
		// pause process step if button is pushed
		IF bStartButton THEN
			nInterruptedState := nKEAState;
			nKEAState := E_KEAOperatingState.break;
		//if homing is finished switch to operational
		ELSIF(bSwitchState) THEN
			nKEAState := E_KEAOperatingState.standby;
			bErrorResetHoming := FALSE;
		END_IF
	E_KEAOperatingState.interruption:
		nState := E_SystemOperatingState.working;
		systemState.sOperatingState := 'working';
		localState.sKEAOperatingState := 'working - interruption';
		Operational();
		//if interruption is terminated switch to next step
		IF(NOT bInterruptProcess) THEN
			nKEAState := nInterruptedState + 1;
			tonStepTimer.IN := FALSE;
		END_IF
	E_KEAOperatingState.break:
		nState := E_SystemOperatingState.working;
		systemState.sOperatingState := 'working';	
		localState.sKEAOperatingState := 'working - break';
		Operational(bSwitchToWorking => bSwitchState);
		//if break is terminated switch to next step
		IF bSwitchState THEN
			nKEAState := nStateInBreak;
		END_IF
	E_KEAOperatingState.error:
		nState := E_SystemOperatingState.standby;
		systemState.sOperatingState := 'standby';	
		localState.sKEAOperatingState := 'error';
		flipFlopResetErrors(SET1 := bResetErrors, RESET := (nKEAState = E_KEAOperatingState.error));
		// only start tank heater in ramp-up
		RampUp();
		IF flipFlopResetErrors.Q1 THEN
			bErrorResetHoming := TRUE;
			Homing(bNotOpenDoorAfterHoming := bErrorResetHoming, bHomingFinished => bSwitchState);
			IF bSwitchState THEN
				nKEAState := E_KEAOperatingState.standby;
			ELSE
				nKEAState := E_KEAOperatingState.homing;		
			END_IF
		END_IF
END_CASE
systemState.nOperatingState := nState;
localState.nKEAOperatingState := nKEAState;
interruptProcessState.nInterruptedState := nInterruptedState;
                
END_METHOD

METHOD CheckError : BOOL
  VAR_OUTPUT
    bError : BOOL;
  END_VAR
                  // local errors
S1(SET1 := NOT bEmergencyStopOk, RESET := bResetErrors, Q1 => errorState.bEmergencyStopError);
S2(SET1 := NOT bConditionToStartOk, RESET := bResetErrors, Q1 => errorState.bConditionToStartError);

// subsystem errors
inletAirHeating.CheckError(bError => errorState.bInletAirHeatingSystemError);
tank.CheckError(bError => errorState.bTankHeatingSystemError);

bError := (
	errorState.bEmergencyStopError OR
	errorState.bConditionToStartError OR
	errorState.bInletAirHeatingSystemError OR
	errorState.bTankHeatingSystemError
);

// set global error
bGlobalError := bError;
errorState.bGlobalError := bGlobalError;
CheckError := bError;
                
END_METHOD

METHOD RampUp : BOOL
  VAR_OUTPUT
    bRampUpFinished : BOOL := FALSE;
  END_VAR
                  // turn all cleaning chamber actors off
CleaningChamber.bPumpSupplyOn						:= FALSE;
CleaningChamber.bRotationBasketEnable 				:= FALSE;
CleaningChamber.bRotationBasketDirectionOfRotation 	:= FALSE;
CleaningChamber.bRotationNoozleFrameEnable 			:= FALSE;
CleaningChamber.bExhaustAirFanOn 					:= FALSE;
CleaningChamber.bBlastNoozleTopOn					:= FALSE;
CleaningChamber.bBlastNoozleBottomOn				:= FALSE;

// turn off air heating
inletAirHeating.bSetStatusOnAutomatic := FALSE;

// turn on tank heating
tank.bSetStatusOnAutomatic := TRUE;

// open door if wanted
CleaningChamber.OpenDoor(
	bOpenDoor := bOpenDoor, 
	bInletAirHeaterOnStatus := inletAirHeating.bInletAirHeaterOn, 
	nActiveState := systemState.nOperatingState
);

// if tank heating is finished, ramp-up is finished
IF tank.nTankHeaterState = E_SystemOperatingState.operational THEN
	bRampUpFinished := TRUE;
END_IF
                
END_METHOD

METHOD Operational : BOOL
  VAR_OUTPUT
    bSwitchToWorking : BOOL := FALSE;
  END_VAR
                  // turn all cleaning chamber actors off
CleaningChamber.bPumpSupplyOn						:= FALSE;
CleaningChamber.bRotationBasketEnable 				:= FALSE;
CleaningChamber.bRotationBasketDirectionOfRotation 	:= FALSE;
CleaningChamber.bRotationNoozleFrameEnable 			:= FALSE;
CleaningChamber.bBlastNoozleTopOn					:= FALSE;
CleaningChamber.bBlastNoozleBottomOn				:= FALSE;

// turn off air heating
inletAirHeating.bSetStatusOnAutomatic := FALSE;

// turn on tank heating
tank.bSetStatusOnAutomatic := TRUE;

// open door if wanted
CleaningChamber.OpenDoor(
	bOpenDoor := bOpenDoor, 
	bInletAirHeaterOnStatus := inletAirHeating.bInletAirHeaterOn, 
	nActiveState := systemState.nOperatingState
);

// if start button is pressed and door is closed, start cleaning process 
bSwitchToWorking := (
	bStartButton AND 
	cleaningChamber.bDoorClosed AND
	NOT bGlobalError AND
	tank.fTankTemperature < fTemperatureLimitUpperWorking AND 
	tank.fTankTemperature > fTemperatureLimitLowerWorking
);
                
END_METHOD

METHOD SelectProgram
                  (*Definition der Programmschrittlänge und prozessparameter*)
CASE nSelectProgram OF
	0:
		sActiveProgram := 'manual';	
		fTankTemperatureSetPoint		:= setKEAProgramManual.fTankTemperatureSetPointManual; 			//Bereich: 30...75°C
		fAirHeatingTemperatureSetPoint	:= setKEAProgramManual.fAirHeatingTemperatureSetPointManual; 	//Bereich: 50...110°C
		tDurationSprayCleaning			:= DINT_TO_TIME(1000*INT_TO_DINT(setKEAProgramManual.nDurationSprayCleaningManual));	//Bereich: 0...300 Sekunden - Zeit für Schrittkette
		tDurationDripping				:= DINT_TO_TIME(1000*INT_TO_DINT(setKEAProgramManual.nDurationDrippingManual));			//Bereich: 0...300 Sekunden - Zeit für Schrittkette
		tDurationSuction				:= DINT_TO_TIME(1000*INT_TO_DINT(setKEAProgramManual.nDurationSuctionManual));			//Bereich: 0...300 Sekunden - Zeit für Schrittkette
		tDurationBlowing				:= DINT_TO_TIME(1000*INT_TO_DINT(setKEAProgramManual.nDurationBlowingManual));			//Bereich: 0...300 Sekunden - Zeit für Schrittkette
		tDurationConvectionDrying		:= DINT_TO_TIME(1000*INT_TO_DINT(setKEAProgramManual.nDurationConvectionDryingManual));	//Bereich: 0...300 Sekunden - Zeit für Schrittkette	
		fTankHeaterHysteresisWidth		:= setKEAProgramManual.fTankHeaterHysteresisWidthManual;		// Definiert Range der Tankheizung
		fTemperatureLimitLowerWorking 	:= setKEAProgramManual.fTemperatureLimitLowerWorking;
		fTemperatureLimitUpperWorking 	:= setKEAProgramManual.fTemperatureLimitUpperWorking;
		bProgramWithBasketRotation		:= setKEAProgramManual.bProgramWithBasketRotation;		// Keine Korbrotation
		sTypeWorkpiece					:= setKEAProgramManual.sTypeWorkpiece;
		fMassWorkpiece					:= setKEAProgramManual.fMassWorkpiece;		// mass in kg	
	1:
		sActiveProgram := 'ArePron';
		fTankTemperatureSetPoint		:= 60; 			//Bereich: 30...75°C
		fAirHeatingTemperatureSetPoint	:= 110; 		//Bereich: 50...110°C
		tDurationSprayCleaning			:= T#600S;		//Bereich: 0...300 Sekunden - Zeit für Schrittkette
		tDurationDripping				:= T#10S;		//Bereich: 0...300 Sekunden - Zeit für Schrittkette
		tDurationSuction				:= T#10S;		//Bereich: 0...300 Sekunden - Zeit für Schrittkette
		tDurationBlowing				:= T#10S;		//Bereich: 0...300 Sekunden - Zeit für Schrittkette
		tDurationConvectionDrying		:= T#90S;		//Bereich: 0...300 Sekunden - Zeit für Schrittkette	
		fTankHeaterHysteresisWidth		:= 2;			// Definiert Range der Tankheizung
		fTemperatureLimitLowerWorking 	:= 55;
		fTemperatureLimitUpperWorking 	:= 65;
		bProgramWithBasketRotation		:= FALSE;		// Keine Korbrotation
		sTypeWorkpiece					:= 'Control plate';
		fMassWorkpiece					:= 0.262;		// mass in kg
	2:
		sActiveProgram := 'Schaumparty';
		fTankTemperatureSetPoint		:= 55; 			//Bereich: 30...75°C
		fAirHeatingTemperatureSetPoint	:= 110; 		//Bereich: 50...110°C
		tDurationSprayCleaning			:= T#240S;		//Bereich: 0...300 Sekunden - Zeit für Schrittkette
		tDurationDripping				:= T#10S;		//Bereich: 0...300 Sekunden - Zeit für Schrittkette
		tDurationSuction				:= T#10S;		//Bereich: 0...300 Sekunden - Zeit für Schrittkette
		tDurationBlowing				:= T#10S;		//Bereich: 0...300 Sekunden - Zeit für Schrittkette
		tDurationConvectionDrying		:= T#60S;		//Bereich: 0...300 Sekunden - Zeit für Schrittkette	
		fTankHeaterHysteresisWidth		:= 4;			// Definiert Range der Tankheizung	
		fTemperatureLimitLowerWorking 	:= 50;
		fTemperatureLimitUpperWorking 	:= 65;
		bProgramWithBasketRotation		:= FALSE;		// Keine Korbrotation
		sTypeWorkpiece					:= 'Control plate';
		fMassWorkpiece					:= 0.262;		// mass in kg
	3:
		sActiveProgram := 'Phi-Abschlussdemo';	
		fTankTemperatureSetPoint		:= 60; 			//Bereich: 30...75°C
		fAirHeatingTemperatureSetPoint	:= 110; 		//Bereich: 50...110°C
		tDurationSprayCleaning			:= T#30S;		//Bereich: 0...300 Sekunden - Zeit für Schrittkette
		tDurationDripping				:= T#10S;		//Bereich: 0...300 Sekunden - Zeit für Schrittkette
		tDurationSuction				:= T#10S;		//Bereich: 0...300 Sekunden - Zeit für Schrittkette
		tDurationBlowing				:= T#11S;		//Bereich: 0...300 Sekunden - Zeit für Schrittkette
		tDurationConvectionDrying		:= T#41S;		//Bereich: 0...300 Sekunden - Zeit für Schrittkette	
		fTankHeaterHysteresisWidth		:= 5;			// Definiert Range der Tankheizung
		fTemperatureLimitLowerWorking 	:= 55;
		fTemperatureLimitUpperWorking 	:= 65;
		bProgramWithBasketRotation		:= FALSE;		// Keine Korbrotation	
		sTypeWorkpiece					:= 'none';
		fMassWorkpiece					:= 0;		// mass in kg
	4:
		sActiveProgram := 'MaschinenTestlauf';	
		fTankTemperatureSetPoint		:= 60; 			//Bereich: 30...75°C
		fAirHeatingTemperatureSetPoint	:= 110; 		//Bereich: 50...110°C
		tDurationSprayCleaning			:= T#5S;		//Bereich: 0...300 Sekunden - Zeit für Schrittkette
		tDurationDripping				:= T#5S;		//Bereich: 0...300 Sekunden - Zeit für Schrittkette
		tDurationSuction				:= T#5S;		//Bereich: 0...300 Sekunden - Zeit für Schrittkette
		tDurationBlowing				:= T#5S;		//Bereich: 0...300 Sekunden - Zeit für Schrittkette
		tDurationConvectionDrying		:= T#5S;		//Bereich: 0...300 Sekunden - Zeit für Schrittkette	
		fTankHeaterHysteresisWidth		:= 5;			// Definiert Range der Tankheizung
		fTemperatureLimitLowerWorking 	:= 55;
		fTemperatureLimitUpperWorking 	:= 70;
		bProgramWithBasketRotation		:= TRUE;		// Korbrotation	
		sTypeWorkpiece					:= 'none';
		fMassWorkpiece					:= 0;		// mass in kg	
	5:
		sActiveProgram := 'CPSL_Testlauf';	
		fTankTemperatureSetPoint		:= 60; 			//Bereich: 30...75°C
		fAirHeatingTemperatureSetPoint	:= 110; 		//Bereich: 50...110°C
		tDurationSprayCleaning			:= T#45S;		//Bereich: 0...300 Sekunden - Zeit für Schrittkette
		tDurationDripping				:= T#5S;		//Bereich: 0...300 Sekunden - Zeit für Schrittkette
		tDurationSuction				:= T#5S;		//Bereich: 0...300 Sekunden - Zeit für Schrittkette
		tDurationBlowing				:= T#5S;		//Bereich: 0...300 Sekunden - Zeit für Schrittkette
		tDurationConvectionDrying		:= T#30S;		//Bereich: 0...300 Sekunden - Zeit für Schrittkette	
		fTankHeaterHysteresisWidth		:= 5;			// Definiert Range der Tankheizung
		fTemperatureLimitLowerWorking 	:= 55;
		fTemperatureLimitUpperWorking 	:= 70;
		bProgramWithBasketRotation		:= FALSE;		// Korbrotation	
		sTypeWorkpiece					:= 'Control plate';
		fMassWorkpiece					:= 0.262;		// mass in kg
	6:
		sActiveProgram := 'Phi720ohneKorb';	
		fTankTemperatureSetPoint		:= 60; 			//Bereich: 30...75°C
		fAirHeatingTemperatureSetPoint	:= 110; 		//Bereich: 50...110°C
		tDurationSprayCleaning			:= T#450S;		//Bereich: 0...300 Sekunden - Zeit für Schrittkette
		tDurationDripping				:= T#25S;		//Bereich: 0...300 Sekunden - Zeit für Schrittkette
		tDurationSuction				:= T#25S;		//Bereich: 0...300 Sekunden - Zeit für Schrittkette
		tDurationBlowing				:= T#70S;		//Bereich: 0...300 Sekunden - Zeit für Schrittkette
		tDurationConvectionDrying		:= T#90S;		//Bereich: 0...300 Sekunden - Zeit für Schrittkette	
		fTankHeaterHysteresisWidth		:= 4;			// Definiert Range der Tankheizung
		fTemperatureLimitLowerWorking 	:= 55;
		fTemperatureLimitUpperWorking 	:= 70;
		bProgramWithBasketRotation		:= FALSE;		// Korbrotation	
		sTypeWorkpiece					:= 'Control plate';
		fMassWorkpiece					:= 0.262;		// mass in kg
END_CASE
                
END_METHOD

METHOD SetStates
                  // set control state
controlState.bStatusOn := bStatusOn;

// set program state
programState.sActiveProgram					:= sActiveProgram;
programState.fTankTemperatureSetPoint		:= fTankTemperatureSetPoint;
programState.fTankHeaterHysteresisWidth 	:= fTankHeaterHysteresisWidth;
programState.fAirHeatingTemperatureSetPoint	:= fAirHeatingTemperatureSetPoint;
programState.nDurationSprayCleaning			:= DINT_TO_INT(TIME_TO_DINT(tDurationSprayCleaning) / 1000);
programState.nDurationDripping				:= DINT_TO_INT(TIME_TO_DINT(tDurationDripping) / 1000);
programState.nDurationSuction				:= DINT_TO_INT(TIME_TO_DINT(tDurationSuction) / 1000);
programState.nDurationBlowing				:= DINT_TO_INT(TIME_TO_DINT(tDurationBlowing) / 1000);
programState.nDurationConvectionDrying 		:= DINT_TO_INT(TIME_TO_DINT(tDurationConvectionDrying) / 1000);
programState.bProgramWithBasketRotation 	:= bProgramWithBasketRotation;
programState.fMassWorkpiece					:= fMassWorkpiece;
programState.sMassWorkpieceUnit				:= 'kg';
programState.sTypeWorkpiece					:= sTypeWorkpiece;
programState.sDurationUnit					:= 's';

// set local state
// sKEAOperatingState and nKEAOperatingState are set in SystemFlowControl
localState.nWorkpieces		:= nWorkpieces;
localState.fCurrent 		:= fCurrent;
localState.fRealPower 		:= fRealPower;
localState.fReactivePower 	:= fReactivePower;
localState.fFrequency 		:= fFrequency;

// set interrupt process state
// nInterruptedState is set in SystemFlowControl
interruptProcessState.fMachinePowerConsumption := fRealPower;
interruptProcessState.stepPowerConsumption.fPowerConsumptionBlowing := 980;
interruptProcessState.stepPowerConsumption.fPowerConsumptionSprayCleaning := 3430;
interruptProcessState.stepPowerConsumption.fPowerConsumptionConvectionDrying := 9350;
interruptProcessState.stepPowerConsumption.fPowerConsumptionDripping := 200;
interruptProcessState.stepPowerConsumption.fPowerConsumptionSuction := 550;
interruptProcessState.stepPowerConsumption.fPowerConsumptionHoming := 250;
interruptProcessState.stepPowerConsumption.fPowerConsumptionOperational := 200;
interruptProcessState.sPowerUnit := 'W';
interruptProcessState.fInterruptionCountdown := TIME_TO_REAL(tTimeToNextInterruption) / 1000;
interruptProcessState.fInterruptionCountdownUnit := 's';
interruptProcessState.stepDuration.fDurationSprayCleaning := TIME_TO_REAL(tDurationSprayCleaning) / 1000;
interruptProcessState.stepDuration.fDurationDripping := TIME_TO_REAL(tDurationDripping) / 1000;
interruptProcessState.stepDuration.fDurationSuction := TIME_TO_REAL(tDurationSuction) / 1000;
interruptProcessState.stepDuration.fDurationBlowing	:= TIME_TO_REAL(tDurationBlowing) / 1000;
interruptProcessState.stepDuration.fDurationConvectionDrying := TIME_TO_REAL(tDurationConvectionDrying) / 1000;
interruptProcessState.stepDuration.sDurationUnit := 's';
interruptProcessState.stepEnergyConsumption.fEnergyConsumptionSprayCleaning := (
	interruptProcessState.stepPowerConsumption.fPowerConsumptionSprayCleaning * interruptProcessState.stepDuration.fDurationSprayCleaning / 3600);
interruptProcessState.stepEnergyConsumption.fEnergyConsumptionConvectionDrying := (
	interruptProcessState.stepPowerConsumption.fPowerConsumptionConvectionDrying * interruptProcessState.stepDuration.fDurationConvectionDrying / 3600);
interruptProcessState.sEnergyUnit := 'Wh';
                
END_METHOD

METHOD TimeToNextInterruption : BOOL
  VAR_INPUT
    nKEAState : E_KEAOperatingState;
    tStepElapsedTime : TIME;
  END_VAR
                  CASE nKEAState OF
	E_KEAOperatingState.operational:
		tTimeToNextInterruption := T#0S;
	E_KEAOperatingState.sprayCleaning:
		tTimeToNextInterruption := tDurationSprayCleaning - tStepElapsedTime + tDurationDripping + tDurationSuction + tDurationBlowing;
	E_KEAOperatingState.dripping:
		tTimeToNextInterruption := tDurationDripping - tStepElapsedTime + tDurationSuction + tDurationBlowing;
	E_KEAOperatingState.suction:
		tTimeToNextInterruption := tDurationSuction - tStepElapsedTime + tDurationBlowing;
	E_KEAOperatingState.blowing:
		tTimeToNextInterruption := tDurationBlowing - tStepElapsedTime;
	E_KEAOperatingState.convectionDrying:
		tTimeToNextInterruption := tDurationConvectionDrying - tStepElapsedTime;
END_CASE
	
	
                
END_METHOD

METHOD SelectInterruptionMode : BOOL
                  //enable interruption of process is in algorithm or manual mode 
IF control.bManualModeActivated THEN
	bInterruptProcess := interruptProcess.bInterruptProcessManual;
ELSIF control.bAlgorithmModeActivated AND bAlgorithmPermission THEN
	bInterruptProcess := interruptProcess.bInterruptProcessAlgorithm;
ELSE
	bInterruptProcess := FALSE;
END_IF
                
END_METHOD
END_FUNCTION_BLOCK

{attribute 'symbol' := 'none'}
FUNCTION_BLOCK FB_ActorContinous EXTENDS FB_Actor2Point IMPLEMENTS ITF_ActorContinous
  VAR_INPUT
    fSetPointAutomatic : REAL;  (* unit depending setpoint *)
  END_VAR
  VAR_OUTPUT
    fOperatingPoint : REAL;  (* unit depending operating point *)
  END_VAR
  VAR
    {attribute 'symbol' := 'readwrite'}
    setSetPoint : ST_SetSetPoint;
    {attribute 'symbol' := 'readwrite'}
    setPointState : ST_SetPointState;
    fSetPoint : REAL;  (* actual set setpoint *)
    aSetPointLimits : ARRAY[1..2] OF REAL;  (* control mode and unit depending setpoint limits that are set by abstract method SetSetPointLimits() in a subclass *)
  END_VAR

            
          

METHOD SelectControlMode : BOOL
                  SUPER^.SelectControlMode();

//add changing set point to method
IF control.bManualModeActivated THEN
	fsetPoint := setSetPoint.fSetPointManual;
ELSIF control.bAlgorithmModeActivated AND bAlgorithmPermission THEN
	fsetPoint := setSetPoint.fSetPointAlgorithm;
ELSE
	fsetPoint := fSetPointAutomatic;
END_IF
                
END_METHOD

METHOD SetPointCheck : BOOL
                  fSetPoint := MAX(fSetPoint, aSetPointLimits[1]);
fSetPoint := MIN(fSetPoint, aSetPointLimits[2]);
                
END_METHOD

METHOD MAIN : BOOL
                  SelectControlMode();
SetSetPointLimits();
SetPointCheck();
                
END_METHOD

METHOD SetSetPointLimits : BOOL
                  
                
END_METHOD
END_FUNCTION_BLOCK

{attribute 'symbol' := 'none'}
FUNCTION_BLOCK FB_TankSystem EXTENDS FB_SystemContinous IMPLEMENTS ITF_System
  VAR_INPUT
    nActiveState : E_SystemOperatingState := E_SystemOperatingState.standby;
    fTankHeaterHysteresisWidth : REAL := 4;
    bGlobalError : BOOL;
    bResetErrors : BOOL;
    fTemperatureLimitLowerWorking : REAL := 55;
    fTemperatureLimitUpperWorking : REAL := 65;
  END_VAR
  VAR_OUTPUT
    nTankHeaterState : E_SystemOperatingState := E_SystemOperatingState.standby;
    fTankTemperature : REAL;
  END_VAR
  VAR
    {attribute 'symbol' := 'readwrite'}
    tankHeater : FB_Actor2Point;  (* actors *)
    bSupplyFreshWaterOn : BOOL;
    bOilSeparationOn : BOOL;
    {attribute 'symbol' := 'readwrite'}
    tankTempSensor : ST_TempSensorState;  (* sensors *)
    bFilterMonitor : BOOL;
    bTankLevelMin : BOOL;
    bTankLevelNominal : BOOL;
    bTankLevelMax : BOOL;
    bOilSeparationLevelMax : BOOL;
    bDemineralOk : BOOL;
    {attribute 'symbol' := 'readwrite'}
    localState : ST_TankState;  (* states *)
    {attribute 'symbol' := 'readwrite'}
    errorState : ST_TankErrorState;
    {attribute 'symbol' := 'readwrite'}
    storeEnergyInherentlyState : ST_StoreEnergyInherentlyState;
    bSetStatusOnTankHeater : BOOL := TRUE;  (* internal variables *)
    bAlgorithmPermissionTankHeater : BOOL := TRUE;
    fTemperatureLimitLowerCritical : REAL := 8;
    fTemperatureLimitUpperCritical : REAL := 85;
  END_VAR

            MAIN();
ReadInputs();
CheckAlgorithmPermission(fTemperatureOffset := 1);

// instantiate tank heater
tankHeater(
	bSetStatusOnAutomatic 	:= bSetStatusOnTankHeater AND NOT bGlobalError,
	bAlgorithmPermission 	:= bAlgorithmPermissionTankHeater
);

// turn on fresh water if not in error and tank level is not nominal and if in working
bSupplyFreshWaterOn := NOT bGlobalError AND NOT bTankLevelNominal AND nActiveState = E_SystemOperatingState.working;

// control oil separation
bOilSeparationOn := OilSeparation();

// set states
SetStates();

// set local outputs
nTankHeaterState := systemState.nOperatingState;

SetOutputs();

          

METHOD ReadInputs : BOOL
                  // read tank temperature
PRG_AnalogInputs(tankTempSensor => tankTempSensor);
fTankTemperature := tankTempSensor.fValue;

// read inputs
bFilterMonitor 			:= inputs.bFilterMonitor;
bTankLevelMin 			:= NOT inputs.bTankLevelMin_NOT;
bTankLevelNominal		:= NOT inputs.bTankLevelNominal_NOT;
bTankLevelMax			:= NOT inputs.bTankLevelMax_NOT;
bOilSeparationLevelMax 	:= inputs.bOilSeparationLevelMax;
bDemineralOk 			:= inputs.bDemineralOk;
                
END_METHOD

METHOD SetOutputs : BOOL
                  // set ouputs
outputs.bTankHeatingOn 		:= tankHeater.bStatusOn;
outputs.bSupplyFreshWaterOn := bSupplyFreshWaterOn;
outputs.bOilSeparationOn 	:= bOilSeparationOn;
                
END_METHOD

METHOD CheckError : BOOL
  VAR_OUTPUT
    bError : BOOL;
  END_VAR
                  T1(IN := bTankLevelMin, PT := T#3S);
S1(SET1 := T1.Q, RESET := bResetErrors, Q1 => errorState.bErrorTankLevelLow);

T2(IN := bTankLevelMax, PT := T#3S);
S2(SET1 := T2.Q, RESET := bResetErrors, Q1 => errorState.bErrorTankLevelFull);

T3(IN := NOT bDemineralOk AND bSupplyFreshWaterOn, PT := T#5S);
S3(SET1 := T3.Q, RESET := bResetErrors, Q1 => errorState.bErrorFreshWaterSupply);

T4(IN := fTankTemperature < fTemperatureLimitLowerCritical, PT := T#1S);
S4(SET1 := T4.Q, RESET := bResetErrors, Q1 => errorState.bErrorTankTemperatureCriticalLow);

T5(IN := fTankTemperature > fTemperatureLimitUpperCritical, PT := T#1S);
S5(SET1 := T5.Q, RESET := bResetErrors, Q1 => errorState.bErrorTankTemperatureCriticalHigh);

bError := (
	errorState.bErrorTankLevelLow OR
	errorState.bErrorTankLevelFull OR
	errorState.bErrorFreshWaterSupply OR
	errorState.bErrorTankTemperatureCriticalLow OR 
	errorState.bErrorTankTemperatureCriticalHigh
);
CheckError := bError;
                
END_METHOD

METHOD RampUp : BOOL
  VAR_OUTPUT
    bRampUpFinished : BOOL := FALSE;
  END_VAR
                  // turn tank heater on for warm-up
IF fTankTemperature < fTemperatureLimitLowerWorking THEN
	bSetStatusOnTankHeater := TRUE;
	bRampUpFinished := FALSE;
ELSE
	bRampUpFinished := TRUE;
END_IF

                
END_METHOD

METHOD OilSeparation : BOOL
  VAR
    Biestable_RS_hysteresis : RS;
  END_VAR
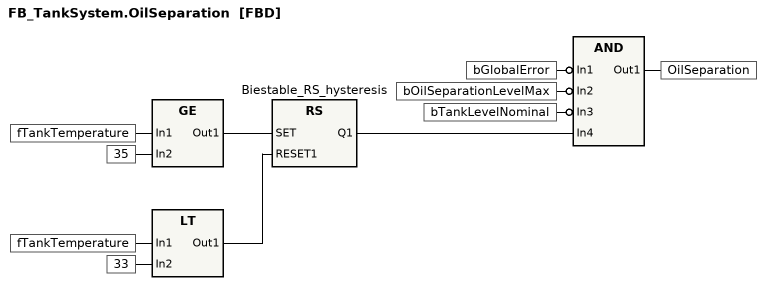
(* FBD diagram, written out as Structured Text *)
Biestable_RS_hysteresis(SET := fTankTemperature >= 35, RESET1 := fTankTemperature < 33);
OilSeparation := NOT bGlobalError AND NOT bOilSeparationLevelMax AND NOT bTankLevelNominal AND Biestable_RS_hysteresis.Q1;
END_METHOD

METHOD CtrlTankHeater : BOOL
  VAR_INPUT
    fTankTemperature : REAL;
    fTemperatureLimitLower : REAL;
    fTemperatureLimitUpper : REAL;
  END_VAR
  VAR
    nTankTemperature : INT;
    nTemperatureLimitLower : INT;
    nTemperatureLimitUpper : INT;
    fConversionFactor : REAL := 100;
  END_VAR
                  // convert real to int with conversion factor
nTankTemperature 		:= REAL_TO_INT(fTankTemperature * fConversionFactor);
nTemperatureLimitLower 	:= REAL_TO_INT(fTemperatureLimitLower * fConversionFactor);
nTemperatureLimitUpper 	:= REAL_TO_INT(fTemperatureLimitUpper * fConversionFactor);

hysteresis(
	IN := nTankTemperature,
	HIGH := nTemperatureLimitUpper,
	LOW := nTemperatureLimitLower,
	OUT => CtrlTankHeater
);
                
END_METHOD

METHOD Working : BOOL
  VAR_OUTPUT
    bSwitchToOperational : BOOL := FALSE;
  END_VAR
                  // control tank heater in hysteresis in automatic mode
bSetStatusOnTankHeater := CtrlTankHeater(
	fTankTemperature := tankTempSensor.fValue,
	fTemperatureLimitLower := fSetPoint - fTankHeaterHysteresisWidth / 2,
	fTemperatureLimitUpper := fSetPoint + fTankHeaterHysteresisWidth / 2
);

                
END_METHOD

METHOD SetSetPointLimits : BOOL
  VAR
    fTemperatureLimitLower : REAL;
    fTemperatureLimitUpper : REAL;
  END_VAR
                  CASE systemState.nOperatingState OF
	E_SystemOperatingState.standby, E_SystemOperatingState.rampUp, E_SystemOperatingState.rampDown:
		fTemperatureLimitLower := fTemperatureLimitLowerCritical + fTankHeaterHysteresisWidth / 2;
		fTemperatureLimitUpper := fTemperatureLimitUpperCritical - fTankHeaterHysteresisWidth / 2;
	E_SystemOperatingState.operational, E_SystemOperatingState.working:
		fTemperatureLimitLower := fTemperatureLimitLowerWorking + fTankHeaterHysteresisWidth / 2;
		fTemperatureLimitUpper := fTemperatureLimitUpperWorking - fTankHeaterHysteresisWidth / 2;
END_CASE

aSetPointLimits[1] := fTemperatureLimitLower;
aSetPointLimits[2] := fTemperatureLimitUpper;
setPointState.aSetPointLimits := aSetPointLimits;
                
END_METHOD

METHOD SetStates : BOOL
                  // set control state
controlState.bStatusOn := bStatusOn;

// set set point state
setPointState.aSetPointLimits 		:= aSetPointLimits;
setPointState.fSetPoint 			:= fSetPoint;
setPointState.fOperatingPoint 		:= fOperatingPoint;
setPointState.sSetPointUnit 		:= 'degreeC';
setPointState.sOperatingPointUnit 	:= 'degreeC';

// set local state
localState.bTankHeatingOn						:= tankHeater.bStatusOn;
localState.bSupplyFreshWaterOn					:= bSupplyFreshWaterOn;
localState.bOilSeparationOn 					:= bOilSeparationOn;
localState.fTankTemperature 					:= fTankTemperature;
localState.bFilterMonitor 						:= bFilterMonitor;
localState.bTankLevelMin 						:= bTankLevelMin;
localState.bTankLevelNominal					:= bTankLevelNominal;
localState.bTankLevelMax						:= bTankLevelMax;
localState.bOilSeparationLevelMax 				:= bOilSeparationLevelMax;
localState.bDemineralOk 						:= bDemineralOk;
localState.fTankHeaterHysteresisWidth 			:= fTankHeaterHysteresisWidth;
localState.fTemperatureLimitLowerWorking 		:= fTemperatureLimitLowerWorking;
localState.fTemperatureLimitUpperWorking 		:= fTemperatureLimitUpperWorking;
localState.fTemperatureLimitLowerCritical 		:= fTemperatureLimitLowerCritical;
localState.fTemperatureLimitUpperCritical 		:= fTemperatureLimitUpperCritical;
localState.sTemperatureUnit						:= 'degreeC';
localState.fCleaningFluidSpecificHeatCapacity	:= 4190;
localState.sCleaningFluidSpecificHeatCapacityUnit := 'J/(kg*K)';
localState.fCleaningFluidDensity				:= 1000;
localState.sCleaningFluidDensityUnit			:= 'kg/m^3';
localState.fTankVolume							:= 0.320;
localState.sTankVolumeUnit						:= 'm^3';

// set store energy inherently state
storeEnergyInherentlyState.fNominalLoad 			:= 10000;
storeEnergyInherentlyState.sPowerUnit				:= 'W';
storeEnergyInherentlyState.sMachineStateCorrelation := 'standby, operational, working';
storeEnergyInherentlyState.sProcessStepCorrelation 	:= 'sprayCleaning; dripping; suction; blowing; convectionDrying; homing';
storeEnergyInherentlyState.bOperatingPoint			:= tankHeater.bStatusOn;
storeEnergyInherentlyState.fProcessValue			:= fTankTemperature;
storeEnergyInherentlyState.aFlexibilityLimits		:= setPointState.aSetPointLimits;
storeEnergyInherentlyState.sProcessValueUnit		:= 'degreeC';
                
END_METHOD

METHOD CheckAlgorithmPermission : BOOL
  VAR_INPUT
    fTemperatureOffset : REAL;
  END_VAR
                  // give algorithm permission to control tank heater if temperature is inside the limits
IF (
	bAlgorithmPermissionTankHeater AND 
	(aSetPointLimits[1] <= tankTempSensor.fValue) AND 
	(tankTempSensor.fValue <= aSetPointLimits[2]) AND 
	NOT bGlobalError
) THEN
	bAlgorithmPermissionTankHeater := TRUE;
// if permission is denied reset permission if inside the limits with offset
ELSIF (
	NOT bAlgorithmPermissionTankHeater AND 
	(aSetPointLimits[1] + fTemperatureOffset <= tankTempSensor.fValue) AND 
	(tankTempSensor.fValue <= aSetPointLimits[2] - fTemperatureOffset) AND 
	NOT bGlobalError
) THEN
	bAlgorithmPermissionTankHeater := TRUE;
ELSE
	bAlgorithmPermissionTankHeater := FALSE;
END_IF
                
END_METHOD

METHOD Standby : BOOL
                  bSetStatusOnTankHeater 	:= FALSE;
bSupplyFreshWaterOn		:= FALSE;
bOilSeparationOn		:= FALSE;
                
END_METHOD
END_FUNCTION_BLOCK

{attribute 'symbol' := 'none'}
FUNCTION_BLOCK FB_SystemContinous EXTENDS FB_ActorContinous IMPLEMENTS ITF_System, ITF_ActorContinous
  VAR
    {attribute 'symbol' := 'readwrite'}
    systemState : ST_SystemState;
  END_VAR

            
          

METHOD MAIN : BOOL
                  SUPER^.MAIN();
SystemFlowControl();
                
END_METHOD

METHOD SystemFlowControl : INT
                  CheckError(bError => bSystemError);
systemState.bError := bSystemError;

IF NOT bSystemError THEN
	CASE nState OF
		E_SystemOperatingState.standby:
			systemState.sOperatingState := 'standby';
			bSwitchState := FALSE;
			Standby();
			//if turned on switch to ramp-up
			IF(bSetStatusOn) THEN
				nState := E_SystemOperatingState.rampUp;
			END_IF
		E_SystemOperatingState.rampUp:
			systemState.sOperatingState := 'ramp-up';
			RampUp(bRampUpFinished => bSwitchState);
			//if turned off switch to ramp-down
			IF(NOT bSetStatusOn) THEN
				nState := E_SystemOperatingState.rampDown;
			//if ramp-up finished switch to operational
			ELSIF(bSwitchState) THEN
				nState := E_SystemOperatingState.operational;
			END_IF
		E_SystemOperatingState.operational:
			systemState.sOperatingState := 'operational';
			Operational(bSwitchToWorking => bSwitchState);
			//if turned off switch to ramp-down
			IF(NOT bSetStatusOn) THEN
				nState := E_SystemOperatingState.rampDown;
			//switch to working if desired
			ELSIF(bSwitchState) THEN
				nState := E_SystemOperatingState.working;
			END_IF
		E_SystemOperatingState.working:
			systemState.sOperatingState := 'working';
			Working(bSwitchToOperational => bSwitchState);
			//if turned off switch to ramp-down
			IF(NOT bSetStatusOn) THEN
				nState := E_SystemOperatingState.rampDown;
			//switch to operational if desired
			ELSIF(bSwitchState) THEN
				nState := E_SystemOperatingState.operational;
			END_IF
		E_SystemOperatingState.rampDown:
			systemState.sOperatingState := 'ramp-down';
			RampDown(bRampDownFinished => bSwitchState);
			//if turned on switch to ramp-up
			IF(bSetStatusOn) THEN
				nState := E_SystemOperatingState.rampUp;
			//if ramp-down finished switch to standby
			ELSIF(bSwitchState) THEN
				nState := E_SystemOperatingState.standby;
			END_IF
	END_CASE
ELSE
	RampDown(bRampDownFinished => bSwitchState);
	IF bSwitchState THEN
		systemState.sOperatingState := 'standby';
		nState := E_SystemOperatingState.standby;
	ELSE
		systemState.sOperatingState := 'ramp-down';	
		nState := E_SystemOperatingState.rampDown;		
	END_IF
	
END_IF
systemState.nOperatingState := nState;
                
END_METHOD

METHOD SetSetPointLimits : BOOL
                  
                
END_METHOD

METHOD CheckError : BOOL
  VAR_OUTPUT
    bError : BOOL;
  END_VAR
                  bError := FALSE;
                
END_METHOD

METHOD Operational : BOOL
  VAR_OUTPUT
    bSwitchToWorking : BOOL := FALSE;
  END_VAR
                  // basic implementation sets ouput true such that this step is skipped
bSwitchToWorking := TRUE;
                
END_METHOD

METHOD RampDown : BOOL
  VAR_OUTPUT
    bRampDownFinished : BOOL := FALSE;
  END_VAR
                  // basic implementation sets ouput true such that this step is skipped
bRampDownFinished := TRUE;
                
END_METHOD

METHOD RampUp : BOOL
  VAR_OUTPUT
    bRampUpFinished : BOOL := FALSE;
  END_VAR
                  // basic implementation sets ouput true such that this step is skipped
bRampUpFinished := TRUE;
                
END_METHOD

METHOD Working : BOOL
  VAR_OUTPUT
    bSwitchToOperational : BOOL := FALSE;
  END_VAR
                  // basic implementation is empty such that system stays in working
                
END_METHOD

METHOD Standby : BOOL
                  // basic implementation is empty
                
END_METHOD
END_FUNCTION_BLOCK

{attribute 'symbol' := 'none'}
FUNCTION_BLOCK FB_InletAirHeatingSystem EXTENDS FB_SystemContinous IMPLEMENTS ITF_System
  VAR_INPUT
    bGlobalError : BOOL;
    bResetErrors : BOOL;
  END_VAR
  VAR_OUTPUT
    bAirSupplyFlowOk : BOOL;  (* safety sensor *)
    bInletAirHeaterOn : BOOL;  (* state of heating *)
  END_VAR
  VAR
    {attribute 'symbol' := 'readwrite'}
    inletAirHeater : FB_Actor2Point;  (* actors *)
    bInletAirFanOn : BOOL;
    bOpenInletAirShutOffValve : BOOL;
    {attribute 'symbol' := 'readwrite'}
    airSupplyTempSensor : ST_TempSensorState;  (* sensors *)
    bInletAirShutOffValveOpen : BOOL;
    bInletAirShutOffValveClosed : BOOL;
    bAirSupplyTempSensorOk : BOOL;
    {attribute 'symbol' := 'readwrite'}
    errorState : ST_InletAirHeatingErrorState;  (* states *)
    {attribute 'symbol' := 'readwrite'}
    localState : ST_InletAirHeatingState;
    {attribute 'symbol' := 'readwrite'}
    storeEnergyInherentlyState : ST_StoreEnergyInherentlyState;
    fAirSupplyTemperature : REAL;  (* internal variables *)
    fTemperatureLimitLowerCritical : REAL := 5;
    fTemperatureLimitUpperCritical : REAL := 150;
  END_VAR

            MAIN();
ReadInputs();

// instantiate inlet air heater
inletAirHeater(bAlgorithmPermission := NOT CheckError());
bInletAirHeaterOn := inletAirHeater.bStatusOn;

// read air supply temperature
PRG_AnalogInputs(airSupplyTempSensor => airSupplyTempSensor);
fAirSupplyTemperature := airSupplyTempSensor.fValue;

// set states
SetStates();

SetOutputs();
          

METHOD SetOutputs : BOOL
                  // set ouputs
outputs.bOpenInletAirShutOffValve 	:= bOpenInletAirShutOffValve;
outputs.bInletAirFanOn 				:= bInletAirFanOn;
outputs.bInletAirHeaterOn			:= inletAirHeater.bStatusOn;
                
END_METHOD

METHOD ReadInputs : BOOL
                  // read inputs
bInletAirShutOffValveOpen 	:= inputs.bInletAirShutOffValveOpen;
bInletAirShutOffValveClosed := inputs.bInletAirShutOffValveClosed;
bAirSupplyTempSensorOk		:= inputs.bAirSupplyTempSensorOk;
bAirSupplyFlowOk 			:= inputs.bAirSupplyFlowOk;
                
END_METHOD

METHOD SetSetPointLimits : BOOL
                  aSetPointLimits[1] := fTemperatureLimitLowerCritical;
aSetPointLimits[2] := fTemperatureLimitUpperCritical;
                
END_METHOD

METHOD CheckError : BOOL
  VAR_OUTPUT
    bError : BOOL;
  END_VAR
                  // error if inlet air shut off valve doesn't open in 5 seconds
T1(
	IN := (bOpenInletAirShutOffValve AND NOT bInletAirShutOffValveOpen) OR (bOpenInletAirShutOffValve AND bInletAirShutOffValveClosed),
	PT := T#5S
);
S1(SET1 := T1.Q, RESET := bResetErrors, Q1 => errorState.bInletAirShutOffValveOpeningError);

// error if inlet air shut off valve doesn't close in 5 seconds
T2(
	IN := (NOT bOpenInletAirShutOffValve AND NOT bInletAirShutOffValveClosed) OR (NOT bOpenInletAirShutOffValve AND bInletAirShutOffValveOpen),
	PT := T#5S
);
S2(SET1 := T2.Q, RESET := bResetErrors, Q1 => errorState.bInletAirShutOffValveClosingError);

// error if inlet air shut off valve sensors are both true
T3(
	IN := (bInletAirShutOffValveClosed AND bInletAirShutOffValveOpen),
	PT := T#1S
);
S3(SET1 := T3.Q, RESET := bResetErrors, Q1 => errorState.bInletAirShutOffValveSensorsError);

// error if air supply temperature sensor is in error
T4(IN := NOT bAirSupplyTempSensorOk, PT := T#1S);
S4(SET1 := T4.Q, RESET := bResetErrors, Q1 => errorState.bAirSupplyTempSensorError);

// error if inlet air supply is not ok in 20 seconds
T5(IN := (bInletAirFanOn AND NOT bAirSupplyFlowOk), PT := T#20S);
S5(SET1 := T5.Q, RESET := bResetErrors, Q1 => errorState.bInletAirFanError);
	
// check air temperature
T6(IN := (fAirSupplyTemperature < fTemperatureLimitLowerCritical), PT := T#1S);
S6(SET1 := T6.Q, RESET := bResetErrors, Q1 => errorState.bErrorAirTemperatureCriticalLow);

T7(IN := (fAirSupplyTemperature > fTemperatureLimitUpperCritical), PT := T#1S);
S7(SET1 := T6.Q, RESET := bResetErrors, Q1 => errorState.bErrorAirTemperatureCriticalHigh);

bError := (
	errorState.bInletAirShutOffValveOpeningError OR 
	errorState.bInletAirShutOffValveClosingError OR
	errorState.bInletAirShutOffValveSensorsError OR
	//errorState.bAirSupplyTempSensorError OR
	errorState.bInletAirFanError OR 
	errorState.bErrorAirTemperatureCriticalLow OR 
	errorState.bErrorAirTemperatureCriticalHigh
);
CheckError := bError;
                
END_METHOD

METHOD RampDown : BOOL
  VAR_OUTPUT
    bRampDownFinished : BOOL := FALSE;
  END_VAR
                  inletAirHeater(bSetStatusOnAutomatic :=FALSE);
bInletAirFanOn :=FALSE;

IF NOT bAirSupplyFlowOk THEN
	bOpenInletAirShutOffValve := FALSE;
END_IF

IF NOT bInletAirShutOffValveOpen AND NOT bAirSupplyFlowOk THEN
	bRampDownFinished := TRUE;
END_IF
                
END_METHOD

METHOD RampUp : BOOL
  VAR_OUTPUT
    bRampUpFinished : BOOL := FALSE;
  END_VAR
                  bOpenInletAirShutOffValve := TRUE;

IF bInletAirShutOffValveOpen THEN
	bInletAirFanOn :=TRUE;
END_IF

IF bInletAirShutOffValveOpen AND bAirSupplyFlowOk THEN
	bRampUpFinished := TRUE;
END_IF
                
END_METHOD

METHOD Working : BOOL
  VAR_OUTPUT
    bSwitchToOperational : BOOL := FALSE;
  END_VAR
                  IF bInletAirShutOffValveOpen AND bAirSupplyFlowOk AND (fAirSupplyTemperature <= (fSetPoint - 5)) THEN
	inletAirHeater(bSetStatusOnAutomatic :=TRUE);
END_IF
		
IF NOT bInletAirShutOffValveOpen OR NOT bAirSupplyFlowOk OR (fAirSupplyTemperature >= fSetPoint)THEN
	inletAirHeater(bSetStatusOnAutomatic :=FALSE);
END_IF
                
END_METHOD

METHOD SetStates : BOOL
                  // set control state
controlState.bStatusOn := bStatusOn;

// set set point state
setPointState.aSetPointLimits 		:= aSetPointLimits;
setPointState.fSetPoint 			:= fSetPoint;
setPointState.fOperatingPoint 		:= fOperatingPoint;
setPointState.sSetPointUnit 		:= 'degreeC';
setPointState.sOperatingPointUnit 	:= 'degreeC';

// set local state
localState.fAirSupplyTemperature 			:= fAirSupplyTemperature;
localState.bInletAirShutOffValveOpen		:= bInletAirShutOffValveOpen;
localState.bInletAirShutOffValveClosed		:= bInletAirShutOffValveClosed;
localState.bAirSupplyTempOk					:= bAirSupplyTempSensorOk;
localState.bAirSupplyFlowOk					:= bAirSupplyFlowOk;
localState.fTemperatureLimitLowerCritical	:= fTemperatureLimitLowerCritical;
localState.fTemperatureLimitUpperCritical	:= fTemperatureLimitUpperCritical;
localState.bInletAirFanStatusOn				:= bInletAirFanOn;

// set store energy inherently state
storeEnergyInherentlyState.fNominalLoad 			:= 8;
storeEnergyInherentlyState.sPowerUnit				:= 'kW';
storeEnergyInherentlyState.sMachineStateCorrelation := 'working';
storeEnergyInherentlyState.sProcessStepCorrelation 	:= 'convectionDrying';
                
END_METHOD

METHOD Standby : BOOL
                  // turn everything off
inletAirHeater(bSetStatusOnAutomatic :=FALSE);
bOpenInletAirShutOffValve 	:= FALSE;
bInletAirFanOn				:= FALSE;
                
END_METHOD
END_FUNCTION_BLOCK

{attribute 'symbol' := 'none'}
FUNCTION_BLOCK FB_CleaningChamberSystem
  VAR_INPUT
    bGlobalError : BOOL;
    bResetErrors : BOOL;
    tMaxDurationExhaustFanOn : TIME;
    bPumpSupplyOn : BOOL;  (* actors *)
    bRotationBasketEnable : BOOL;
    bRotationBasketDirectionOfRotation : BOOL;
    bRotationNoozleFrameEnable : BOOL;
    bExhaustAirFanOn : BOOL;
    bBlastNoozleTopOn : BOOL;
    bBlastNoozleBottomOn : BOOL;
  END_VAR
  VAR_OUTPUT
    bBasketHomed : BOOL;  (* sensors *)
    bNoozleFrameHomed : BOOL;
    bDoorClosed : BOOL;
    bMotorsDrivesOk : BOOL;
    bDoorLoadingSafetyOk : BOOL;
  END_VAR
  VAR
    {attribute 'symbol' := 'readwrite'}
    systemState : ST_SystemState;  (* states *)
    {attribute 'symbol' := 'readwrite'}
    localState : ST_CleaningChamberState;
    {attribute 'symbol' := 'readwrite'}
    errorState : ST_CleaningChamberErrorState;
    bOpenProtectiveDoorLoading : BOOL;  (* local *)
    tonOpenDoorDelay : TON;
    srOpenDoorDelay : SR;
    bDoorOpen : BOOL;
  END_VAR

            ReadInputs();
CheckError(bError => systemState.bError);
// delay of open door
srOpenDoorDelay(SET1 := bDoorOpen, RESET := tonOpenDoorDelay.Q, Q1 => bOpenProtectiveDoorLoading);
tonOpenDoorDelay(IN := bOpenProtectiveDoorLoading, PT := T#2S);
ExhaustFanIfDoorOpen();

SetStates();
SetOutputs();
          

METHOD CtrlBlastNoozles : BOOL
  VAR_INPUT
    tBlastNoozlesPulseDuration : TIME;
    tBlastNoozlesPulsePeriod : TIME;
  END_VAR
  VAR_OUTPUT
    bBlastNoozleBottomOn : BOOL;
    bBlastNoozleTopOn : BOOL;
  END_VAR
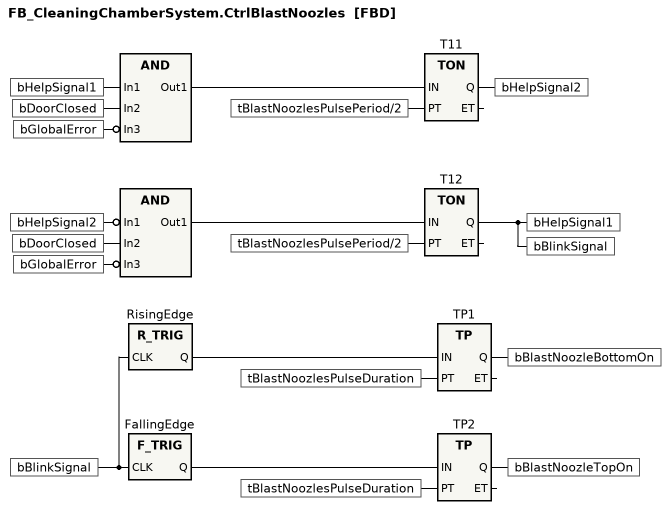
(* FBD diagram, written out as Structured Text *)
T11(IN := bHelpSignal1 AND bDoorClosed AND NOT bGlobalError, PT := tBlastNoozlesPulsePeriod/2);
bHelpSignal2 := T11.Q;
T12(IN := NOT bHelpSignal2 AND bDoorClosed AND NOT bGlobalError, PT := tBlastNoozlesPulsePeriod/2);
bHelpSignal1 := T12.Q;
bBlinkSignal := T12.Q;
RisingEdge(CLK := bBlinkSignal);
TP1(IN := RisingEdge.Q, PT := tBlastNoozlesPulseDuration);
bBlastNoozleBottomOn := TP1.Q;
FallingEdge(CLK := bBlinkSignal);
TP2(IN := FallingEdge.Q, PT := tBlastNoozlesPulseDuration);
bBlastNoozleTopOn := TP2.Q;
END_METHOD

METHOD CheckError : BOOL
  VAR_OUTPUT
    bError : BOOL;
  END_VAR
                  S1(SET1 := NOT bMotorsDrivesOk, RESET := bResetErrors, Q1 => errorState.bMotorsDrivesError);
S2(SET1 := NOT bDoorLoadingSafetyOk, RESET := bResetErrors, Q1 => errorState.bDoorLoadingSafetyError);

bError := errorState.bMotorsDrivesError OR errorState.bDoorLoadingSafetyError;
CheckError := bError;
                
END_METHOD

METHOD OpenDoor : BOOL
  VAR_INPUT
    bOpenDoor : BOOL;
    bInletAirHeaterOnStatus : BOOL;
    nActiveState : E_SystemOperatingState := E_SystemOperatingState.working;
  END_VAR
                  IF(	
	bOpenDoor AND
	nActiveState <> E_SystemOperatingState.working AND
	bEmergencyStopOk AND
	NOT bInletAirHeaterOnStatus AND
	NOT bPumpSupplyOn AND
	NOT bRotationBasketEnable AND
	NOT bRotationNoozleFrameEnable AND
	NOT bBlastNoozleBottomOn AND
	NOT bBlastNoozleTopOn
) THEN
	bDoorOpen := TRUE;
ELSE
	bDoorOpen 			:= FALSE;
	bExhaustAirFanOn	:= FALSE;
END_IF;
                
END_METHOD

METHOD ExhaustFanIfDoorOpen : BOOL
  VAR
    bStartExhaustFan : BOOL;
  END_VAR
                  // set bStartExhaustFan if door is open, reset bStartExhaustFan if door is closed
IF bDoorClosed THEN
	bStartExhaustFan := FALSE;
ELSE
	bStartExhaustFan := TRUE;
END_IF

T1(IN := bStartExhaustFan, PT := tMaxDurationExhaustFanOn);

// operate exhaust fan for tMaxDurationExhaustFanOn if door is open
IF NOT bDoorClosed THEN
	bExhaustAirFanOn := NOT T1.Q;
END_IF

                
END_METHOD

METHOD SetStates : BOOL
                  // set system state
IF(
	bPumpSupplyOn OR
	bRotationBasketEnable OR
	bRotationBasketDirectionOfRotation OR
	bRotationNoozleFrameEnable OR
	bExhaustAirFanOn OR
	bBlastNoozleTopOn OR
	bBlastNoozleBottomOn OR
	bOpenProtectiveDoorLoading
) THEN
	systemState.nOperatingState := E_SystemOperatingState.working;
	systemState.sOperatingState := 'working';
ELSE
	systemState.nOperatingState := E_SystemOperatingState.operational;
	systemState.sOperatingState := 'operational';
END_IF

// set local state
localState.bPumpSupplyStatusOn 					:= bPumpSupplyOn;
localState.bRotationBasketStatusOn 				:= bRotationBasketEnable;
localState.bRotationBasketDirectionOfRotation 	:= bRotationBasketDirectionOfRotation;
localState.bRotationNoozleFrameStatusOn 		:= bRotationNoozleFrameEnable;
localState.bExhaustAirFanStatusOn 				:= bExhaustAirFanOn;
localState.bBlastNoozleTopStatusOn				:= bBlastNoozleTopOn;
localState.bBlastNoozleBottomStatusOn			:= bBlastNoozleBottomOn;
localState.bProtectiveDoorLoadingOpen			:= NOT bDoorClosed;
                
END_METHOD

METHOD ReadInputs : BOOL
                  bBasketHomed 			:= inputs.bBasketHomed;
bNoozleFrameHomed 		:= inputs.bNoozleFrameHomed;
bDoorClosed				:= inputs.bDoorClosed;
bMotorsDrivesOk 		:= inputs.bMotorsDrivesOk;
bDoorLoadingSafetyOk	:= inputs.bDoorLoadingSafetyOk;
                
END_METHOD

METHOD SetOutputs : BOOL
                  // set outputs
outputs.bPumpSupplyOn 						:= bPumpSupplyOn;
outputs.bRotationBasketEnable 				:= bRotationBasketEnable;
outputs.bRotationBasketDirectionOfRotation 	:= bRotationBasketDirectionOfRotation;
outputs.bRotationNoozleFrameEnable 			:= bRotationNoozleFrameEnable;
outputs.bExhaustAirFanOn 					:= bExhaustAirFanOn;
outputs.bBlastNoozleTopOn 					:= bBlastNoozleTopOn;
outputs.bBlastNoozleBottomOn 				:= bBlastNoozleBottomOn;
outputs.bOpenProtectiveDoorLoading			:= bOpenProtectiveDoorLoading;
                
END_METHOD
END_FUNCTION_BLOCK

{attribute 'symbol' := 'none'}
FUNCTION_BLOCK FB_System2Point EXTENDS FB_Actor2Point IMPLEMENTS ITF_System
  VAR
    {attribute 'symbol' := 'readwrite'}
    systemState : ST_SystemState;
  END_VAR

            
          

METHOD RampDown : BOOL
  VAR_OUTPUT
    bRampDownFinished : BOOL := FALSE;
  END_VAR
                  // basic implementation sets ouput true such that this step is skipped
bRampDownFinished := TRUE;
                
END_METHOD

METHOD Operational : BOOL
  VAR_OUTPUT
    bSwitchToWorking : BOOL := FALSE;
  END_VAR
                  // basic implementation sets ouput true such that this step is skipped
bSwitchToWorking := TRUE;
                
END_METHOD

METHOD CheckError : BOOL
  VAR_OUTPUT
    bError : BOOL;
  END_VAR
                  bError := FALSE;
                
END_METHOD

METHOD Working : BOOL
  VAR_OUTPUT
    bSwitchToOperational : BOOL := FALSE;
  END_VAR
                  // basic implementation is empty such that system stays in working
                
END_METHOD

METHOD RampUp : BOOL
  VAR_OUTPUT
    bRampUpFinished : BOOL := FALSE;
  END_VAR
                  // basic implementation sets ouput true such that this step is skipped
bRampUpFinished := TRUE;
                
END_METHOD

METHOD MAIN : BOOL
                  SelectControlMode();
SystemFlowControl();
                
END_METHOD

METHOD SystemFlowControl : INT
                  CheckError(bError => bSystemError);
systemState.bError := bSystemError;

IF NOT bSystemError THEN
	CASE nState OF
		E_SystemOperatingState.standby:
			systemState.sOperatingState := 'standby';
			bSwitchState := FALSE;
			Standby();
			//if turned on switch to ramp-up
			IF(bSetStatusOn) THEN
				nState := E_SystemOperatingState.rampUp;
			END_IF
		E_SystemOperatingState.rampUp:
			systemState.sOperatingState := 'ramp-up';
			RampUp(bRampUpFinished => bSwitchState);
			//if turned off switch to ramp-down
			IF(NOT bSetStatusOn) THEN
				nState := E_SystemOperatingState.rampDown;
			//if ramp-up finished switch to operational
			ELSIF(bSwitchState) THEN
				nState := E_SystemOperatingState.operational;
			END_IF
		E_SystemOperatingState.operational:
			systemState.sOperatingState := 'operational';
			Operational(bSwitchToWorking => bSwitchState);
			//if turned off switch to ramp-down
			IF(NOT bSetStatusOn) THEN
				nState := E_SystemOperatingState.rampDown;
			//switch to working if desired
			ELSIF(bSwitchState) THEN
				nState := E_SystemOperatingState.working;
			END_IF
		E_SystemOperatingState.working:
			systemState.sOperatingState := 'working';
			Working(bSwitchToOperational => bSwitchState);
			//if turned off switch to ramp-down
			IF(NOT bSetStatusOn) THEN
				nState := E_SystemOperatingState.rampDown;
			//switch to operational if desired
			ELSIF(bSwitchState) THEN
				nState := E_SystemOperatingState.operational;
			END_IF
		E_SystemOperatingState.rampDown:
			systemState.sOperatingState := 'ramp-down';
			RampDown(bRampDownFinished => bSwitchState);
			//if turned on switch to ramp-up
			IF(bSetStatusOn) THEN
				nState := E_SystemOperatingState.rampUp;
			//if ramp-down finished switch to standby
			ELSIF(bSwitchState) THEN
				nState := E_SystemOperatingState.standby;
			END_IF
	END_CASE
ELSE
	RampDown(bRampDownFinished => bSwitchState);
	IF bSwitchState THEN
		systemState.sOperatingState := 'standby';
		nState := E_SystemOperatingState.standby;
	ELSE
		systemState.sOperatingState := 'ramp-down';	
		nState := E_SystemOperatingState.rampDown;		
	END_IF
	
END_IF
systemState.nOperatingState := nState;
                
END_METHOD

METHOD Standby : BOOL
                  // basic implementation is empty
                
END_METHOD
END_FUNCTION_BLOCK
